(* CODESYS project MQTT 1.1.0.4.library
   Description: MQTT Stuff
      Using some cool stuff of OSCAT libs.
      see oscat.de
      
      more to describe
   Version: 1.1.0.4
   Title: MQTT
   Author: Stefan Dreyer
   DocFormat: reStructuredText
   Placeholder: SD_MQTT
   LanguageModelAttribute: qualified-access-only
   DefaultNamespace: SD_MQTT
   Company: Stefan Dreyer

Project tree, tasks and I/O mapping:
  libraries: Standard, * (System); Time and Date, 3.5.7.0 (3S - Smart Software Solutions GmbH); 3S Storage, 3.5.13.0 (3S - Smart Software Solutions GmbH); SysMem, 3.5.12.0 (System); SysTypes2 Interfaces, 3.5.4.0 (System); CmpErrors2 Interfaces, 3.5.15.0 (System); CAA Memory, 3.5.12.0 (CAA Technical Workgroup); BASIC, 3.5.16.0 (OSCAT); Common Helper for development, 1.0.0.2 (Stefan Dreyer); NETWORK, * (OSCAT)
  MQTT/
    Function Blocks/
      function block HANDLE_MQTT [ST]: ResetPingTime, MakePingPaket, StateMashineOut, StateMashineIn, BuildPublishPaket, MoveBufferForSplitPaket, BuildSubscribePaket, BuildUnsubscribePaket, SendOutData, SendInData, ParseIncoming, ParseIncomingPublish, CheckLenghtBuffer, FB_Exit, destroy, OutputPublish, MergeSplitedPublish, Publish, PublishSendDone, PushError
      function block MQTT_CONTROL [ST]
      function block MQTTPublish [ST]
      function block MQTTBase [ST]: SetMqttInOut
      function block MQTTSubscribe [ST]
      function block InsertSplitTopic [ST]: reset
      function block HandleSplitTopic [ST]: FullInit, LowInit, destroy, GetSplitTopic, FB_Exit, NewTopic, PushSplitLevel, DestroyOldSplit, CheckTopicMatchToMe, CheckTopicValid
      function block InsertSplitPayload [ST]: reset
      function block MQTTValue [ST]: Init
      function block MQTTState [ST]: Init
      function block MQTTPushover [ST]
      CallbackFBs/
        SingelCallbacks/
          function block SingelStringCallback [ST]: PublishReceived, Init, ResetReceived
          function block AllValuesCallback [ST]: PublishReceived, Init, ResetReceived
        ListCallbacks/
          function block ListStringCallback [ST]: PublishReceived, InitAsSplitTopic, InitAsSplitPayload
          function block ListAllValuesCallback [ST]: PublishReceived, InitAsSplitTopic, InitAsSplitPayload
        Callback Collector/
          function block CallbackCollector [ST]: put, PublishReceived, destroy, FB_Exit
          function block ReceiveValueWithStrucur [ST]: InitReceiveStructur
          function block ReceiveValue [ST]: PublishReceived, initAsFindPayload, initAsFindTopic, makePointer, initAsFindTopicAndPayload, SetOutput, initAsFindLastTopic
          function block ReceiveString [ST]: PublishReceived, initAsFindTopic, initAsFindPayload
          function block ReceiverBase [ST]: init, CheckMatch, GetValue
    Function/
      function InsertStringToBufferAndLength [ST]
      function DoRemainingLength [ST]
      function GetRemainingLength [ST]
      function CheckTopicLevel [ST]
      function DoRemainingLengthBevor [ST]
      function InitMQTTValue [ST]
    Structs/
      data type MQTT_IN_OUT
      data type DATA_FROM_BROKER
      data type MQTT_INFO
      data type MQTT_COM
      data type DATA_TO_BROKER
      data type MQTT_IN_DATA
      data type PAKET_DATA
      data type MQTT_OUT_DATA
      data type REMAINING_LENGTH_RETURN
      data type SPLIT_TOPIC
      data type SEND_INFOS
      data type RECEIVE_PAKET
      data type COM_CONFIG
      data type PUSHOVER_DATA
      CallbackStuff/
        data type MQTT_SUBSCRIBE_CALLBACKS
        data type LIST_STRING_CALLBACK_DATA
        data type CALLBACK_DATA
        data type LIST_ALLVALUES_CALLBACK_DATA
        data type CALLBACK_INSTANCES
      data type ONE_ERROR
    ENUMs/
      data type MESSAGETYPE
      data type QoS
      data type STEPS_OUT
      data type STEPS_IN
      data type INSERT_SPLIT_RETURN
      data type TOPIC_VALID
      data type TOPIC_MATCH
      data type PROG_NUM
      data type PUSHOVER_SOUND
      data type ERRORS
      data type RECEIVER_INIT_TYPS
      data type RECEIVE_TYPS
    Global Constants/
      global variables MyConstants
    global variables GVL_MQTT
    TestCases/
      function block TestcaseCheckTopivValid [ST]
      function block TestSubscribeOld [ST]
      function block TestMqtt [ST]
      function block TestMqttTLS [ST]
      function block TestTopicMatch [ST]
      function block TestPublishValue [ST]
      function block testHighReceive [ST]
      function block testHighReceiveSplitPayload [ST]
      function block HighLoadPublish [ST]
      function block testHighLoadPublish [ST]
      Test Interfaces/
        function block FooBarReceivingFB [ST]: PublishReceived, initAsFindTopic, getLastTreeName, initAsFindPayload
        function block exampleForFbs [ST]
        function block TestCallbackCollecktor [ST]: FB_Exit
      function block TestLongPublish [ST]
      function block TestLongStringList [ST]
      function block TestStringPointer [ST]
      function block TestUserPassword [ST]
      function block TestMemHandle [ST]
      function block TestSplitTopic [ST]
      function block testLongTime [ST]
    Docs/
      program Doku [ST]
    Exampels/
      function block TestOutOfTheBoxNoTLS [ST]
      function block TestOutOfTheBoxTLS [ST]
    Interfaces/
      interface MQTT_SUBSCRIBE_CALLBACK: PublishReceived
*)

// MQTT/Structs/MQTT_IN_OUT
TYPE MQTT_IN_OUT :
STRUCT
	//pointer to handle FB
	handleFB:POINTER TO HANDLE_MQTT;
	In: POINTER TO PAKET_DATA;
	//in free, true if free
	InFree: BOOL := TRUE;
	//time, date, impulse...
	TDI : CommonTypesAndFunctions.TIME_DATE_IMPULS_DATA;
	//TLS stuff data
	TLS_CONFIG : POINTER TO CommonTypesAndFunctions.TLS_CONFIG := 0;
	
	BROKER_CONNECTED:BOOL;
	//config for boot up
	COM_CONFIG:COM_CONFIG;
	(*client ID, only chars 0123456789abcdefghijklmnopqrstuvwxyzABCDEFGHIJKLMNOPQRSTUVWXYZ"
	System never can be anonymos
	*)
	ClientID:STRING(23):='CODESYS_MQTT';
	BuildWillTopicAndMessage: BOOL := TRUE;
	WillTopicBase:STRING(255) := 'MQTTWill';
	ClientWillTopic:STRING(255) := 'DEAD';
	ClientWillMessage:STRING(30) := 'DIED';
	//usage of dynamic RAM
	dynMemUsage:UDINT;
	{info 'TODO implement!'}
	(*set this to one if you want the client to act like the standardt says
	if set to one and we receve mor publish pakets than we can handle, QoS 0 packets are lost
	and QoS 1 and 2 packets have to be repeaded by he broker*)
	disconnectOnBufferOverflow:BOOL;
	//do you want the Reorderevents in the history?
	putReordersInHistory:BOOL := FALSE;
	//Log buffer Moves?
	LogBufferMoves:BOOL;
END_STRUCT
END_TYPE

// MQTT/ENUMs/MESSAGETYPE
TYPE MESSAGETYPE :
(
	CONNECT 	:= 16#10,
	CONNACK 	:= 16#20,
	PUBLISH 	:= 16#30,
	PUBACK 		:= 16#40,
	PUBREC		:= 16#50,
	PUBREL		:= 16#60,
	PUBCOMP		:= 16#70,
	SUBSCRIBE 	:= 16#80,
	SUBACK 		:= 16#90,
	UNSUBSCRIBE := 16#A0,
	UNSUBACK 	:= 16#B0,
	PINGREQ 	:= 16#C0,
	PINGRESP	:= 16#D0,
	DISCONNECT 	:= 16#E0
) BYTE;
END_TYPE

// MQTT/ENUMs/QoS
TYPE QoS :
(
	AtMostOnce:= 2#0,
	AtLeastOnce:= 2#1,
	ExactlyOnce:= 2#10,
	Fail:=2#10000000
) BYTE;
END_TYPE

// MQTT/Structs/DATA_FROM_BROKER
TYPE DATA_FROM_BROKER :
STRUCT
	//use array in size of network buffer to split message dynamic, maybe not ... best is dynamic mammory....
	//or use an array of Pointer....
	//or callbacks
	// so lets try to buffer public messages and releas one per cycle to application...
	//now we try dynamic memmory....
	//MQTT Topic from Broker
	MqttTopic:POINTER TO STRING;
	Topics:POINTER TO SPLIT_TOPIC;
	//MQTT Payload for Broker
	//Payload from broker --> Pointer
	MqttPayload:POINTER TO BYTE;
	//Payload size
	MqttPayloadSize:UDINT;
	//MQTT Message Type
	MessageType:MESSAGETYPE;
	//Data received
	DataReceived:BOOL;
	
END_STRUCT
END_TYPE

// MQTT/Structs/MQTT_INFO
TYPE MQTT_INFO :
STRUCT
	MQTT_CONNECTED : BOOL;
	MQTT_ERROR : STRING(OSCAT_BASIC.STRING_LENGTH);
END_STRUCT
END_TYPE

// MQTT/Structs/MQTT_COM
(*contro struct between HANDLE_MQTT and MQTT_CONTROL*)
TYPE MQTT_COM :
STRUCT
	S_BUF : NETWORK_BUFFER;
	R_BUF : NETWORK_BUFFER;
	MQTT_CON : BOOL;//if falling edge close with disconnect packet
	MQTT_ABORT :BOOL;//if using this to disconnect, don't send disconnect paket....
	MQTT_URL : STRING(OSCAT_BASIC.STRING_LENGTH);
	MQTT_PACKET_NO : WORD;
	TIMEOUT : TIME;
	//DNS_IP4 : DWORD;
	//set to true if you want to use TLS
	TLS: BOOL;
	//data to TLS stuff
	TLS_CONFIG:POINTER TO CommonTypesAndFunctions.TLS_CONFIG := 0;
	(*
	0= non
	1= received
	2= error*)
	MQTT_RCV_STATE : BYTE;
	ERROR_C : DWORD;
	ERROR_T : BYTE;
	//CONNECT_TO_LOCALHOST:BOOL;
	CLIENT_ID:STRING(23);
	CLIENT_WILL_TOPIC:STRING(255);//Topic vof will message after client id
	CLIENT_WILL_MESSAGE_DEAD:STRING(255);
	{info 'implement parameter'}
	CLIENT_WILL_RETAIN:BOOL:=TRUE;
	//pakte wihout request-- return to receive state 1
	MQTT_NO_AWNSER: BOOL;


END_STRUCT
END_TYPE

// MQTT/Structs/DATA_TO_BROKER
TYPE DATA_TO_BROKER :

STRUCT
	//Data of Paket
	PaketData:PAKET_DATA;
END_STRUCT
END_TYPE

// MQTT/Structs/MQTT_IN_DATA
TYPE MQTT_IN_DATA :
STRUCT
	step:STEPS_IN;
	PaketID:WORD;
	WaitsForBuffFree:ULINT;
	TimeOut:ton;
	TimeOutStarted:BOOL;
	PUBLISHOrder:UINT;
	PUBCOMPOrder:UINT;
	QoS:QoS;
	CountPubrecRepeat:UINT;;
END_STRUCT
END_TYPE

// MQTT/Structs/PAKET_DATA
TYPE PAKET_DATA :
STRUCT
	//MQTT Topic for Broker
	MqttTopic:POINTER TO STRING;
	//Topic length
	MqttTopicLength:UINT;
	//MQTT Payload for Broker
	MqttPayload:POINTER TO BYTE;
	//Payload length
	MqttPayloadLength:UDINT;
	//MQTT Message Type
	MessageType:MESSAGETYPE;
	//MQTT QoS
	MessageQoS:QoS;
	//SUCACK QoS Response
	SubackQoS:QoS;
	//MQTT reatin
	MessageRetain:BOOL;
	//Retry of paket
	DUP: BOOL;
	//PakatID for header
	PaketId:WORD;
	//ID of MQTT FB to store or of request to Broker
	//FbId:UINT;
	//Send was succsessfull
	SendSucsess: BOOL;
	//Callback FB for subscription
	Callback:MQTT_SUBSCRIBE_CALLBACK;
	//split topic for subscribe
	SplitTopic:POINTER to HandleSplitTopic; 
	//errore registering the callback
	CallbackError: BOOL;
	//Expecting String
	ExpectingString: BOOL;


	
END_STRUCT
END_TYPE

// MQTT/Structs/MQTT_OUT_DATA
TYPE MQTT_OUT_DATA :
STRUCT
	InDataFromFb: POINTER TO PAKET_DATA;
	step:STEPS_OUT;
	WaitsForBuffFree:ULINT;
	PUBRECOrder:UINT;
	TimeOut:ton;
	TimeOutStarted:BOOL;
	PUBLISHOrder:UINT;
	PUBRELRepeatCounter:UINT;
END_STRUCT
END_TYPE

// MQTT/ENUMs/STEPS_OUT
{attribute 'qualified_only'}
{attribute 'strict'}
TYPE STEPS_OUT :
(
	WAIT_DATA := 0, SEND_PUBLSIH, WAIT_PUBREC, SEND_PUBREL,
	WAIT_PUBCOMP, WAIT_PUBACK, WAIT_PINGRESP, SEND_SUBSCRIBE, 
	WAIT_SUBACK, SEND_UNSUBSCRIBE, WAIT_UNSUBACK
);
END_TYPE

// MQTT/ENUMs/STEPS_IN
{attribute 'qualified_only'}
{attribute 'strict'}
TYPE STEPS_IN :
(
	WAIT_DATA := 0, SEND_PUBACK, SEND_PUBREC, 
	WAIT_PUBREL, SEND_PUBCOMP
);
END_TYPE

// MQTT/Structs/REMAINING_LENGTH_RETURN
TYPE REMAINING_LENGTH_RETURN :
STRUCT
	RemainingLength:UDINT;
	IndexAfterRemainingLength:UINT; 
	Error:BOOL;
	//not all bytes of remaining length in buffer...
	BuffToSmall:BOOL;
	//size of remaining length
	SizeRemainingLength:USINT;
	
END_STRUCT
END_TYPE

// MQTT/Structs/SPLIT_TOPIC
TYPE SPLIT_TOPIC :
STRUCT
	//this is going to be a pointer to a array of pointer to stings  
	Topics:POINTER TO POINTER TO STRING;
	//count of vailid fields in the array
	ValidFields:UINT;
	
END_STRUCT
END_TYPE

// MQTT/ENUMs/INSERT_SPLIT_RETURN
{attribute 'qualified_only'}
{attribute 'strict'}
TYPE INSERT_SPLIT_RETURN :
(
	INSERT_NOT_VALID := 0, INSERT_DONE , INSERT_PENDING, INSERT_ERROR
);
END_TYPE

// MQTT/ENUMs/TOPIC_VALID
{attribute 'qualified_only'}
{attribute 'strict'}
TYPE TOPIC_VALID :
(
	TOPIC_UNTESTED := 0, TOPIC_VALID := 2, TOPIC_NOT_VALID := 1, TOPIC_NO_TEST := 3
)BYTE;
END_TYPE

// MQTT/ENUMs/TOPIC_MATCH
{attribute 'qualified_only'}
{attribute 'strict'}
TYPE TOPIC_MATCH :
(
	TOPIC_MATCHES := 1, TOPIC_DONT_MATCHES := 2, TOPIC_NO_MEMORY := 3
)BYTE;
END_TYPE

// MQTT/Structs/SEND_INFOS
TYPE SEND_INFOS :
STRUCT
		
//this index is to be subscribed
	SubscribeIndex:UINT;
	SubscribeNeeded:BOOL := FALSE;
	SubscribeBlocking: BOOL;

	//this index is to be subscribed
	
	UnsubscribeIndex:UINT;
	UnsubscribeNeeded:BOOL := FALSE;
	UnsubscribeBlocking: BOOL;

	//this index is to be published
	PublishBlocking: BOOL;
	PublishBlockingIndex : UINT;

	//this index is to be published
	PingIndex:UINT;
	PingNeeded: BOOL;
	
END_STRUCT
END_TYPE

// MQTT/Structs/RECEIVE_PAKET
//used for test cases...
TYPE RECEIVE_PAKET :
STRUCT
	//MQTT Topic
	MqttTopic:STRING(2000);
	//MQTT Payload
	MqttPayload:STRING(2000);
END_STRUCT
END_TYPE

// MQTT/ENUMs/PROG_NUM
{attribute 'qualified_only'}
{attribute 'strict'}
TYPE PROG_NUM :
(
	Publish, Subscribe, ParseIncomming, MoveBuffer, ParsePublish, GetBufferFreePos, GetSplitTopic, DESTROY_HANDLE_MQTT,
	DESTROY_SPLIT_TOPIC, STATE_MASHINE_IN,  STATE_MASHINE_OUT, SendOutData, SendInData, SendOutDataInsertTopic, SendOutDataInsertPayload,
	DESTROY_SPLIT_TOPIC_DONE, DESTROY_HANDLE_MQTT_DONE, DESTROY_CALLBACK_COLLECTOR, DESTROY_CALLBACK_COLLECTOR_DONE
);
END_TYPE

// MQTT/Structs/COM_CONFIG
(*here the maximum sizes of paylod and topics are defined
if dynamic low init of split topic is used, don't care about MaxTopicElementSize*)
TYPE COM_CONFIG :
STRUCT
	//max payload size
	MaxPayloadSize : UDINT := 2000;
	//max topic levels
	MaxTopicLevels:UINT := 25;
	//Max Topic elemt size
	MaxTopicElementSize:UINT:=255;
	
END_STRUCT
END_TYPE

// MQTT/Structs/PUSHOVER_DATA
TYPE PUSHOVER_DATA :
STRUCT
	Trigger:POINTER TO BOOL;
	Topic:POINTER TO STRING;
	Payload:POINTER TO STRING;
	Prio:USINT;
	Sound:PUSHOVER_SOUND;
	IsConfig:BOOL;
	R_T:R_TRIG;
	NeedToPush:BOOL;
	Negate:BOOL;
END_STRUCT
END_TYPE

// MQTT/ENUMs/PUSHOVER_SOUND
{attribute 'qualified_only'}
{attribute 'strict'}
TYPE PUSHOVER_SOUND :
(
	Standart := 1
);
END_TYPE

// MQTT/Structs/CallbackStuff/MQTT_SUBSCRIBE_CALLBACKS
TYPE MQTT_SUBSCRIBE_CALLBACKS :
STRUCT
	Callback:MQTT_SUBSCRIBE_CALLBACK;
	//expecting string
	ExpectingString: BOOL;
	SplitTopic:POINTER TO HandleSplitTopic;
	//set to false if slot is aquired by an subscription
	free:BOOL:=TRUE;
	
END_STRUCT
END_TYPE

// MQTT/Structs/CallbackStuff/LIST_STRING_CALLBACK_DATA
TYPE LIST_STRING_CALLBACK_DATA :
STRUCT
	//pointer to target string
	Target:POINTER TO STRING;
	//pointer to last subtopic or Payload Data to compare with
	SubTopic:POINTER TO STRING;

END_STRUCT
END_TYPE

// MQTT/Structs/CallbackStuff/CALLBACK_DATA
(*this data is passed to a subscription callback*)

TYPE CALLBACK_DATA :
STRUCT
	{info 'make size check due use of memmove...'}
	(*the Payload String,
	be aware, this pointer will only copy 255 bytes. If more needed, use memmove!*)
	PayloadString:POINTER TO STRING(255);
	(*pointer to binary payload*)
	Payload:POINTER TO BYTE;
	(*size of binary payload*)
	PayloadSize:UDINT;
	(*here you get the compleete received topic string, maybe bigger then 255 byte!*)
	TopicOut:POINTER TO STRING(255);
	//split topic....
	TopicOutSplit:POINTER TO SPLIT_TOPIC;
	//Payload is string
	PayloadIsString: BOOL;

END_STRUCT
END_TYPE

// MQTT/Structs/CallbackStuff/LIST_ALLVALUES_CALLBACK_DATA
TYPE LIST_ALLVALUES_CALLBACK_DATA :
STRUCT
	VarTYPE:CommonTypesAndFunctions.VAR_TYPES;
	Target:CommonTypesAndFunctions.ALL_TYPES_UNION_POINTER;
	//pointer to last subtopic or Payload Data to compare with
	SubTopic:POINTER TO STRING;
END_STRUCT
END_TYPE

// MQTT/Structs/CallbackStuff/CALLBACK_INSTANCES
{attribute 'enable_dynamic_creation'} 
TYPE CALLBACK_INSTANCES :
STRUCT
	callback:MQTT_SUBSCRIBE_CALLBACK;
	next: POINTER TO CALLBACK_INSTANCES := 0;
	

END_STRUCT
END_TYPE

// MQTT/Structs/ONE_ERROR
TYPE ONE_ERROR :
STRUCT
	error:ERRORS;
	when:DT;
	ERROR_C : DWORD;
	ERROR_T : BYTE;
	text:STRING(255);
	MqttsDoneIo:ULINT;
	SendetBytes:ULINT;
	ReceivedBytes:ULINT;
END_STRUCT
END_TYPE

// MQTT/ENUMs/ERRORS
{attribute 'qualified_only'}
{attribute 'strict'}
TYPE ERRORS :
(
	NOT_VALID := 0,
	CONNECTION_REFUSED := 1, MAX_PING_REPEATS := 2,
	RECEIVED_PUBISH_TO_BIG_FOR_BUFFER := 3, FULL_PACKET_NOT_RECEIVED := 4,
	RECEIVED_PUBLISH_REMAINING_LENGTH_ERROR := 5,
	NO_MORE_RECEIVE_SLOTS_FREE := 6,
	CONNECTION_ESTABLISHED := 7, TIMEOUT_CONNECTION := 8,
	REPEAT_PUBLISH_PUBCOMP := 9, REPEAT_PUBREL := 10, 
	REORDER_PUBREC := 11, REORDER_PUBLISH_OUTGOING := 12,
	REPEAT_PUBLISH_PUBREC := 13, REPEAT_PUBLISH_PUBACK := 14,
	HARD_DISCONNECT := 15, MOVED_TO_BIG_RECEIVE_BUFFER := 16,
	NEED_BUFFER_MOV := 17, UNKNOWN_PAKET_RECEIVED := 18,
	TO_BIG_PAKET := 19, TOPIC_MOVED_DOWN := 20,
	TOPIC_AND_PAYLOAD_MOVED := 21, PAYLOAD_MOVED_UP := 22,
	TOPIC_MOVED_DOWN_NETWORK := 23, PAYLOAD_MOVED_UP_NETWORK := 24,
	REPEAT_PUBREC := 25, PUBREC_DISCHARGE := 26,
	REODER_PUBLISH_INCOMMING := 27, REORDER_PUBCOMP := 28,
	UNKNOWN_PAKET_IN_MQTT_IN_OUT := 29,
	PUBLISH_NO_SLOT_FREE := 30, OUT_OFF_DYN_MEMORY := 31
);
END_TYPE

// MQTT/ENUMs/RECEIVER_INIT_TYPS
{attribute 'qualified_only'}
{attribute 'strict'}
TYPE RECEIVER_INIT_TYPS :
(
	(*searching for full matching topic*)
	FIND_FULL_TOPIC := 0,
	(*searching for match of last topic*) 
	FIND_LAST_TOPIC,
	(*searching on paylod, from start, spared with delimiter*) 
	FIND_PAYLOAD,
	(*search full topic and one JSON element*)
	JSON_FULL,
	(*searching for last topic and one JSON element*)
	JSON_SMALL,
	(*search with MQTT string(including +, #)*)
	MQTT_STRING,
	(*search with MQTT string(including +, #), then JSON*)
	MQTT_STRING_JSON
);
END_TYPE

// MQTT/ENUMs/RECEIVE_TYPS
{attribute 'qualified_only'}
{attribute 'strict'}
TYPE RECEIVE_TYPS :
(
	FIND_PAYLOAD := 0, FIND_TOPIC := 1, FIND_LAST_TOPIC := 2, FIND_LAST_TOPIC_AND_PAYLOAD := 3 
);
END_TYPE

// MQTT/Global Constants/MyConstants
{attribute 'qualified_only'}
VAR_GLOBAL CONSTANT
	//count of simultanus packets workt on
	IN_OUT_SLOTS_SIZE:UINT:=50;
	NETWORK_BUFFER_LONG_SIZE:UINT:=4095;
	KEEP_ALIVE_TIME : DWORD := 8;
	SENDING_TIMEOUT : TIME := T#4S;
	REPEAT_TIMEOUT : TIME := T#2S;
	REORDER_VALUE :UINT:=50000;//50000
	SUBSTRACTION_VALUE:UINT:=30000;//20000
	MAX_PUBREL_REPEATS : UINT :=10;
END_VAR

// MQTT/GVL_MQTT
{attribute 'qualified_only'}
VAR_GLOBAL
	//Last Progamm stat for debug timeout exception
	ProgNum:PROG_NUM;
	//LOG_BUFFER_MOVES:BOOL;
END_VAR

// MQTT/Function Blocks/HANDLE_MQTT
(*
var/log/mosquitto/mosquitto.log
Messsages are not beeing repeatet, if timout for an answer then connection is canceled, new established and the publisher have to start new
Start the command line subscriber:
mosquitto_sub -v -t 'test/topic'
mosquitto_sub -v -h test.mosquitto.org -t 'test/topic'


sudo apt-get install tshark 

tshark -i 1 -a duration:60 -w /tmp/wlan.pcap

debug / logging :
mosquitto_sub -v -t '$SYS/#'
sudo nano /etc/mosquitto/mosquitto.conf  --> 'log_type all'
Publish test message with the command line publisher:
mosquitto_pub -t 'test/topic' -m 'helloWorld'
change check free to InFbNo

kopieren
sudo cp /var/log/mosquitto/mosquitto.log /tmp/
zugriff
sudo chmod -v a=r /tmp/mosquitto.log


TODO: Take care of clean session, is enabled, do it paramable?
	
*)


FUNCTION_BLOCK HANDLE_MQTT  
VAR_IN_OUT
	
	MQTT_IN_OUT:MQTT_IN_OUT;
END_VAR
VAR_INPUT
	ENABLE : BOOL;
	//use format: user:password@domain:port
	URL : STRING(OSCAT_BASIC.STRING_LENGTH);
	TIMEOUT : TIME;
	TLS: BOOL;

END_VAR
VAR_OUTPUT
	ERROR_C : DWORD;
	ERROR_T : BYTE;
END_VAR
VAR
	MQTT_INFO : MQTT_INFO;
	DT_MQTT:CommonTypesAndFunctions.TIME_DATE_IMPULS;
	MQTT_CONTROL: MQTT_CONTROL;
	step : INT;
	i1 : UINT;
	
	PingSlot:UINT;
	
	COM: MQTT_COM;
	
	connected: BOOL;

	TimeoutConnection:TON;
		
	MqttsDoneIo:ULINT;
	
	CycleTime:DWORD;
	LastCycleTime:DWORD;
	NextPingTime:CAA.TICK;
	PingTime : CAA.TICK := (MyConstants.KEEP_ALIVE_TIME * 1000) - 6000;//next ping after 6 seconds 
	// Ping was sendet
	PingRequestet: BOOL;
	PingData:DATA_TO_BROKER;
	myFbNo:UINT;
	PubrelOrderIndexCounter:UINT;
	PubcompOrderIndexCounter:UINT;
	
	
	
	//Slots for state masdchien for outgoing packets(to broker)
	OutDataSlots:ARRAY[0..MyConstants.IN_OUT_SLOTS_SIZE] OF MQTT_OUT_DATA;
	//Slots for state masdchien for incomming packets(from broker)
	InDataSlots:ARRAY[0..MyConstants.IN_OUT_SLOTS_SIZE] OF MQTT_IN_DATA;
	PublishSendListCount:UINT;
	PublishSendList:ARRAY[0..MyConstants.IN_OUT_SLOTS_SIZE] OF UINT;
	PubrelSendListCount:UINT;
	PubrelSendList:ARRAY[0..MyConstants.IN_OUT_SLOTS_SIZE] OF UINT;
	PubackSendListCount:UINT;
	PubackSendList:ARRAY[0..MyConstants.IN_OUT_SLOTS_SIZE] OF UINT;
	PubrecSendListCount:UINT;
	PubrecSendList:ARRAY[0..MyConstants.IN_OUT_SLOTS_SIZE] OF UINT;
	PubcompSendListCount:UINT;
	PubcompSendList:ARRAY[0..MyConstants.IN_OUT_SLOTS_SIZE] OF UINT;
	
	//Repeted Publishs
	RepeatedPublish:ULINT;
	//Repeatet publishs afert ot much repeat of pubrel
	RepeatedPublishsAfterPubrel:ULINT;
	//Repeted pubrel
	RepeatedPubrel:ULINT;
	//Repeted Ping
	CountRepeatedPing:ULINT;
	//Repeated pings untill disconnect
	CountRepeatedPingDisconnect:UINT;
	//count of Publishs unacknowledged
	PublishsUnacknowledged:UINT;
	//last part of 255 chars of to big paket topic
	LastToBigTopic:STRING(255);
	//count of to big topics
	CountToBigTopics:ULINT;
	//Cont of ength Error Pakets
	CountLengthErrors:ULINT;
	//Count of repeatet publishs
	CountRepeatPublishReceive:ULINT;
	//Count Received Publishs
	CountReceivedPublishs:ULINT;
	//count sended publishs
	CountSendedPublishs:ULINT;
	//Count of repeated subscribs
	CountRepeatSubscribe:ULINT;
	//Count of repeated unsubscribs
	CountRepeatUnsubscribe:ULINT;
	//Count of repeatet pubrec
	CountRepeatetPubrec:ULINT;
	//Count of OutputPublish calls
	CountOutputPublishCalled:ULINT;
	PUBREC_ERROR_ID_BUFFER:ARRAY[0..PUBREC_ERROR_ID_BUFFER_SIZE -1] OF UINT;
	PUBREC_ERROR_INDEX:UINT;
	//send Publish order Index
	OutgoingPublishOrderIndexCounter:UINT;
	//receive Publish order Index
	IncomingPublishOrderIndexCounter:UINT;
	//Received Pubrel, Paket not found
	CountReceivePubrelUnknown:ULINT;
	//Received Unsuback, Paket not found
	CountReceiveUnsubackUnknown:ULINT;
	//Received Suback, Paket not found
	CountReceiveSubackUnknown:ULINT;
	//Received Puback, Paket not found
	CountReceivePubackUnknown:ULINT;
	//Received Pubrec, Paket not found
	CountReceivePubrecUnknown:ULINT;
	//Received Pubcomp, Paket not found
	CountReceivePubcompUnknown:ULINT;
	SendInfos:SEND_INFOS;
	CountOutSendNotFree:ULINT;
	CountInSendNotFree:ULINT;
	CountCantSendPublishBufferToFull:ULINT;
	CounterPublishSendForMonitor:UINT;
	PublishsSendPerSeconde:UINT;
	CounterPublishReceivedForMonitor:UINT;
	PublishsReceivedPerSeconde:UINT;
	NotKnownPaket:MESSAGETYPE;
	CountUnkownPaket:ULINT;
	LastPaktetForUnkownPaket:MESSAGETYPE;
	HelperLastPaktetForUnkownPaket:MESSAGETYPE;
	CountBufferMoves:ULINT;
	CountNothingSend:ULINT;
	CountConnectAttempt:ULINT;
	//count of topic size exceeded
	CountSplitTopicSizeExceeded:ULINT;
	
	
	CountWaitForRestOfPaket:ULINT;
	CountResetBufferIn:ULINT;
	InBufferMoved:UINT;
	SendFree: BOOL;
	
	MySplitTopic:HandleSplitTopic;
	
	
	InsertSplitTopic:InsertSplitTopic;
	InsertSplitPayload:InsertSplitPayload;
	StepBuildPublish:INT;
	StepBuildSubscribe:INT;
	StepBuildUnsubscribe:INT;
	//use this buffer for received publish packets whos size exceded network buffer Size
	SplitPublishBuffer:POINTER TO BYTE;
	SplitPublishBufferSize:UDINT;
	SplitPublishLength:UDINT;
	//output from buffer Don't write new data!
	MaxPublishPacketSize:UDINT;
	PayloadMemorySize: DWORD;
	
	SubscribeCallbacks:ARRAY[0..CALLBACKS_BUFFER_SIZE - 1] OF MQTT_SUBSCRIBE_CALLBACKS;
	
	TopicMemorySize: DWORD;
	
	COM_CONFIG:COM_CONFIG;

	//publish paket broken, waiting for more data
	PublishSplited: BOOL;
	DoDisconnect: BOOL;
	SendetBytes:ULINT;
	ReceivedBytes:ULINT;
	InSlotsWorking:UINT;
	OutSlotsWorking:UINT;
	SplitPublishBufferAllocationSize:UDINT;
	DynMemUsagePointer : POINTER TO UDINT;
	//callbacks array full
	CallbacksFull: BOOL;

	ErrorHistory:ARRAY[0..COUNT_ERROR_HISTORY]OF ONE_ERROR;
	
	localTdi:CommonTypesAndFunctions.TIME_DATE_IMPULS_DATA;
	
	//Step 10 Init is done:
	StepInitDone: BOOL;

	//Local copy of log buffer moves
	LogBufferMoves: BOOL;

	
END_VAR

VAR CONSTANT
	{info 'make configurable'}
	CALLBACKS_BUFFER_SIZE:UINT:=200;
	RECEIVE_PUBLISH_BUFFER_SIZE : UINT := NETWORK_BUFFER_LONG_SIZE * 2;
	TRANSMIT_BUFFER_SIZE : UINT := NETWORK_BUFFER_LONG_SIZE;
	SIZE_PUBREL:UINT := 4;
	SIZE_UNSUBACK:UINT := 4;
	SIZE_PINGRESP:UINT := 2;
	SIZE_PINGREQ:UINT := 2;
	SIZE_SUBACK:UINT := 5;
	SIZE_PUBACK:UINT := 4;
	SIZE_PUBREC:UINT := 4;
	SIZE_PUBCOMP:UINT := 4;
	SIZE_PAKET_BUFFER_HEADER:UINT := 4;
	PUBREC_ERROR_ID_BUFFER_SIZE:UINT:=100;
	MAX_PING_REPEATS:UINT:=10;
	SPLIT_PUBLISH_BUFFER_ADDITIONAL_RAM:UINT:=17;
	COUNT_MAX_PUBREC_REPEAT_TO_DISCHARGE:UINT:=20;
	COUNT_ERROR_HISTORY:UINT:=1000;
END_VAR

IF MQTT_INFO.MQTT_CONNECTED THEN
	SendFree := COM.S_BUF.SIZE = 0;	
END_IF

LogBufferMoves := MQTT_IN_OUT.LogBufferMoves;

CycleTime := OSCAT_BASIC.T_PLC_MS() - LastCycleTime;
LastCycleTime := OSCAT_BASIC.T_PLC_MS();
//get system time and so one
DT_MQTT(
	TDI_Data:= MQTT_IN_OUT.TDI);
localTdi:= MQTT_IN_OUT.TDI ; 
TimeoutConnection(IN:= step = 10, PT:= T#5S);

CASE step OF

	00:	MQTT_IN_OUT.BROKER_CONNECTED := FALSE;
		IF ENABLE THEN
			MQTT_IN_OUT.handleFB := THIS;
			PingRequestet := FALSE;
			PublishsUnacknowledged := 0;
			PUBREC_ERROR_INDEX := 0;
			CountRepeatedPingDisconnect := 0;
			SendetBytes := 0;
			ReceivedBytes := 0;		
			PublishSplited := FALSE;
			DoDisconnect := FALSE;
			SendInfos.PingNeeded := FALSE;
			SendInfos.SubscribeNeeded := FALSE;
			SendInfos.UnsubscribeNeeded := FALSE;
			StepBuildPublish := 0;
			StepBuildSubscribe := 0;
			StepBuildUnsubscribe := 0;
			InsertSplitTopic.reset();
			InsertSplitPayload.reset();
			CountConnectAttempt := CountConnectAttempt + 1;
			DynMemUsagePointer := ADR(MQTT_IN_OUT.dynMemUsage);
			COM.MQTT_URL := URL;
			COM.TIMEOUT := TIMEOUT;
			COM.CLIENT_ID := MQTT_IN_OUT.ClientID;
			COM.TLS := TLS;
			COM.TLS_CONFIG := MQTT_IN_OUT.TLS_CONFIG;
			ResetPingTime();
			//build will topic
			IF MQTT_IN_OUT.BuildWillTopicAndMessage THEN
				COM.CLIENT_WILL_TOPIC := MQTT_IN_OUT.WillTopicBase;
				COM.CLIENT_WILL_TOPIC := Standard.CONCAT(STR1:= COM.CLIENT_WILL_TOPIC, '/');
				COM.CLIENT_WILL_TOPIC := Standard.CONCAT(STR1:= COM.CLIENT_WILL_TOPIC, STR2:= COM.CLIENT_ID);
				COM.CLIENT_WILL_TOPIC := Standard.CONCAT(STR1:= COM.CLIENT_WILL_TOPIC, '/');
				COM.CLIENT_WILL_TOPIC := Standard.CONCAT(STR1:= COM.CLIENT_WILL_TOPIC, MQTT_IN_OUT.ClientWillTopic);
				COM.CLIENT_WILL_TOPIC := Standard.CONCAT(STR1:= '/', COM.CLIENT_WILL_TOPIC);
				COM.CLIENT_WILL_TOPIC := Standard.CONCAT(STR1:= COM.CLIENT_ID, COM.CLIENT_WILL_TOPIC);
			ELSE
				COM.CLIENT_WILL_TOPIC := MQTT_IN_OUT.ClientWillTopic;
			END_IF
			COM.CLIENT_WILL_MESSAGE_DEAD := MQTT_IN_OUT.ClientWillMessage;
			COM_CONFIG := MQTT_IN_OUT.COM_CONFIG;
			FOR i1 := 0 TO MyConstants.IN_OUT_SLOTS_SIZE - 1 DO
				//reset in slots
				InDataSlots[i1].step := STEPS_IN.WAIT_DATA;
				OutDataSlots[i1].step := STEPS_OUT.WAIT_DATA;
				//reset Timeouts...
				InDataSlots[i1].TimeOutStarted := FALSE;
				OutDataSlots[i1].TimeOutStarted := FALSE;
				InDataSlots[i1].TimeOut(IN:= InDataSlots[i1].TimeOutStarted, PT:= MyConstants.REPEAT_TIMEOUT);
				OutDataSlots[i1].TimeOut(IN:= OutDataSlots[i1].TimeOutStarted, PT:= MyConstants.REPEAT_TIMEOUT);
			END_FOR
			//reset callbacks
			FOR i1 := 0 TO CALLBACKS_BUFFER_SIZE - 1 DO
				SubscribeCallbacks[i1].free := TRUE; 
			END_FOR
			IF  MySplitTopic.FullInit(TopicsLevelInit:= COM_CONFIG.MaxTopicLevels, SplitElementSizeInit:= COM_CONFIG.MaxTopicElementSize, dynMemUsageInit:= ADR(MQTT_IN_OUT.dynMemUsage)) THEN
				
				PayloadMemorySize := COM_CONFIG.MaxPayloadSize;
				{warning disable C0033}
				TopicMemorySize := COM_CONFIG.MaxTopicElementSize * COM_CONFIG.MaxTopicLevels;
				MaxPublishPacketSize := (COM_CONFIG.MaxTopicElementSize * COM_CONFIG.MaxTopicLevels) + PayloadMemorySize;
				SplitPublishBufferAllocationSize := MaxPublishPacketSize + SPLIT_PUBLISH_BUFFER_ADDITIONAL_RAM;
				{info 'semaphore'}
				SplitPublishBuffer  := __NEW(BYTE, SplitPublishBufferAllocationSize);//some additional bytes for paket overhead and termination
				IF SplitPublishBuffer = 0 THEN
					PushError(newError:= ERRORS.OUT_OFF_DYN_MEMORY, text:='No Dyn Memory in Step 00 in Handle' );
					step := 60;
				ELSE
					MQTT_IN_OUT.dynMemUsage := MQTT_IN_OUT.dynMemUsage + SplitPublishBufferAllocationSize;
					{warning restore C0033}
		
					step := 10;
					COM.MQTT_CON := TRUE;
					StepInitDone := TRUE;
					
				END_IF
			ELSE
				PushError(newError:= ERRORS.OUT_OFF_DYN_MEMORY, text:='No Dyn Memory in Step 00 in Handle on create SplitTopic' );
				step := 60;
			END_IF
		END_IF	
	10:	IF MQTT_INFO.MQTT_CONNECTED THEN
			step := 40;
			MQTT_IN_OUT.BROKER_CONNECTED := TRUE;
			PushError(newError:= ERRORS.CONNECTION_ESTABLISHED, text:='');
		END_IF
		IF TimeoutConnection.Q THEN
			PushError(newError:= ERRORS.TIMEOUT_CONNECTION, text:='' );
			step := 0;//reset steps
			destroy();
			
		END_IF
	40:	
		IF PublishSplited THEN
			MergeSplitedPublish(MQTT_IN_OUT:= ADR(MQTT_IN_OUT));
		END_IF	
		ParseIncoming(MQTT_IN_OUT:= ADR(MQTT_IN_OUT));
		PublishSendListCount := 0;
		PubrelSendListCount := 0;
		PubackSendListCount := 0;
		PubrecSendListCount := 0;
		PubcompSendListCount := 0;
		StateMashineIn(MQTT_IN_OUT:= ADR(MQTT_IN_OUT));
		StateMashineOut( MQTT_IN_OUT:= ADR(MQTT_IN_OUT));
		
		SendOutData(MQTT_IN_OUT:= ADR(MQTT_IN_OUT));
		SendInData(MQTT_IN_OUT:= ADR(MQTT_IN_OUT));
	
		IF MQTT_IN_OUT.TDI.IMP THEN
			PublishsSendPerSeconde := CounterPublishSendForMonitor;
			CounterPublishSendForMonitor := 0;
			PublishsReceivedPerSeconde := CounterPublishReceivedForMonitor;
			CounterPublishReceivedForMonitor := 0;
		END_IF
		IF COM.S_BUF.SIZE = 0 THEN
			CountNothingSend := CountNothingSend + 1;
		END_IF
		IF NOT ENABLE THEN 	(* beenden? *)
			step := 50;
			
		END_IF;
		IF DoDisconnect THEN
			DoDisconnect := FALSE;
			//here hard disconnect
			PushError(newError:= ERRORS.HARD_DISCONNECT , text:='');
			COM.MQTT_CON := FALSE; (* MQTT Verbindung beenden *)
			COM.MQTT_ABORT := TRUE;
			MQTT_IN_OUT.BROKER_CONNECTED := FALSE;
			step := 60;
		END_IF

(* ~~~~~~~~~~~~~~~~~~~~~~ *)

50: 
	COM.MQTT_CON := FALSE; (* MQTT Verbindung beenden *)
	MQTT_IN_OUT.BROKER_CONNECTED := FALSE;
	step := 60;//wait for disconnect
60:
	IF MQTT_INFO.MQTT_CONNECTED = FALSE THEN
		destroy();
		step := 0;
		MQTT_IN_OUT.BROKER_CONNECTED := FALSE;
	END_IF
END_CASE;



(* ########################## *)

IF CountRepeatedPingDisconnect > MAX_PING_REPEATS THEN
	DoDisconnect := TRUE;
	IF step = 40 THEN
		PushError(newError:= ERRORS.MAX_PING_REPEATS, text:='');
	END_IF
END_IF


SendetBytes := SendetBytes + COM.S_BUF.SIZE;
MQTT_CONTROL(COM:= COM, INFO:=MQTT_INFO);
ReceivedBytes := ReceivedBytes + COM.R_BUF.SIZE;
ERROR_C := COM.ERROR_C;
ERROR_T := COM.ERROR_T;
//handl ping telegram
IF NextPingTime < TICKS.GetTick(xDummy:= TRUE) AND NOT PingRequestet AND connected THEN
	
	MakePingPaket(MQTT_IN_OUT := MQTT_IN_OUT);
	
END_IF

IF COM.ERROR_T > BYTE#0 THEN  (* FEHLER *)
	DoDisconnect := TRUE;
	MQTT_IN_OUT.BROKER_CONNECTED := FALSE;
	PushError(newError:= ERRORS.CONNECTION_REFUSED, text:='');
END_IF;
//put status to local clients
 

connected := MQTT_IN_OUT.BROKER_CONNECTED;
(* ########################## *)

(* revision history


*)

METHOD ResetPingTime
VAR_INPUT
END_VAR
NextPingTime := PingTime + TICKS.GetTick(xDummy:= TRUE);
CountRepeatedPingDisconnect := 0;
END_METHOD

METHOD MakePingPaket
VAR_INPUT
END_VAR
VAR_IN_OUT
	MQTT_IN_OUT:MQTT_IN_OUT;
END_VAR
IF MQTT_IN_OUT.InFree THEN 
	MQTT_IN_OUT.IN := ADR(PingData); //set request
	PingData.PaketData.MessageType := MESSAGETYPE.PINGREQ;
	MQTT_IN_OUT.InFree := FALSE;
	PingRequestet := TRUE;
END_IF
END_METHOD

METHOD StateMashineOut
VAR_INPUT
	
	//StepData:POINTER TO MQTT_OUT_DATA;
	MQTT_IN_OUT : POINTER TO MQTT_IN_OUT;
END_VAR
VAR
	i:UINT;
	j:UINT;
	tmpLowest:UINT;
	minIndex:UINT;
	UnsubscribeLastHighest : UINT := 16#FFFF;
	SubscribeLastHighest : UINT := 16#FFFF;
//	PublishLastHighest : UINT := 16#FFFF;
//	PubrelLastHighest : UINT := 16#FFFF;
	ReceivePaketID:WORD;
	ReceivePakteType:BYTE;
	TempSlotsWorking:UINT;
	
END_VAR
VAR CONSTANT
	
	
END_VAR
(*need a token for coordinate send of pakets....
prio for Awnser and repeat pakets bevor new publish
dont use token, just send paket with next publish index*)
//get paket id
ReceivePaketID := DWORD_TO_WORD(OSCAT_BASIC.DWORD_OF_BYTE(B3:= 0, B2:= 0, B1:= COM.R_BUF.BUFFER[2], B0:= COM.R_BUF.BUFFER[3]));
ReceivePakteType := COM.R_BUF.BUFFER[0] AND 16#F0; 

GVL_MQTT.ProgNum := PROG_NUM.STATE_MASHINE_OUT;
PublishSendListCount := 0;
PubrelSendListCount := 0;

TempSlotsWorking := 0;
FOR i := 0 TO MyConstants.IN_OUT_SLOTS_SIZE - 1 DO
	//do Timers...
	OutDataSlots[i].TimeOut(IN:= OutDataSlots[i].TimeOutStarted, PT:= MyConstants.REPEAT_TIMEOUT);
	CASE OutDataSlots[i].step OF
		
		STEPS_OUT.WAIT_DATA:
			OutDataSlots[i].TimeOutStarted := FALSE;
			IF NOT MQTT_IN_OUT^.InFree THEN//new Data from FBs
				MQTT_IN_OUT^.InFree := TRUE;
				OutDataSlots[i].InDataFromFb := MQTT_IN_OUT^.In;//set Data
				//Pakte id = slot + 1....
				OutDataSlots[i].InDataFromFb^.PaketId := i + 1;
				CASE OutDataSlots[i].InDataFromFb^.MessageType OF
					MESSAGETYPE.PINGREQ:
						OutDataSlots[i].step := STEPS_OUT.WAIT_PINGRESP;
						SendInfos.PingNeeded := TRUE;
						SendInfos.PingIndex := i;
						PingSlot := i;
					//we only sending one subscription per subscribe paket....
					MESSAGETYPE.SUBSCRIBE:
						//check if we have a slot free for subscription
						FOR j := 0 TO CALLBACKS_BUFFER_SIZE - 1 DO
							IF SubscribeCallbacks[j].free THEN
								OutDataSlots[i].step := STEPS_OUT.SEND_SUBSCRIBE;
								CallbacksFull := FALSE;
								EXIT;
							END_IF
						END_FOR
						IF j = CALLBACKS_BUFFER_SIZE THEN
							//no free slot
							MQTT_IN_OUT^.In^.CallbackError := TRUE;
							CallbacksFull := TRUE;
						END_IF
					MESSAGETYPE.UNSUBSCRIBE:
						OutDataSlots[i].step := STEPS_OUT.SEND_UNSUBSCRIBE;
					ELSE
						PushError(newError:= ERRORS.UNKNOWN_PAKET_IN_MQTT_IN_OUT , text:= CONCAT(STR1:= 'Type:', STR2:= TO_STRING(OutDataSlots[i].InDataFromFb^.MessageType)));
				END_CASE
				
			END_IF
		
		STEPS_OUT.WAIT_PINGRESP:
			IF OutDataSlots[i].TimeOutStarted AND OutDataSlots[i].TimeOut.Q AND NOT SendInfos.PingNeeded THEN
				//timeout, need repead
				SendInfos.PingNeeded := TRUE;
				SendInfos.PingIndex := i;
				CountRepeatedPing := CountRepeatedPing + 1; 
				CountRepeatedPingDisconnect := CountRepeatedPingDisconnect + 1;
				OutDataSlots[i].TimeOutStarted := FALSE;
			END_IF
		STEPS_OUT.SEND_UNSUBSCRIBE:
			//check if my paket ID is the lowest to send it
			IF OutDataSlots[i].InDataFromFb^.PaketId < UnsubscribeLastHighest AND NOT SendInfos.UnsubscribeNeeded THEN
				SendInfos.UnsubscribeIndex := i;
				SendInfos.UnsubscribeNeeded := TRUE;
				UnsubscribeLastHighest := OutDataSlots[i].InDataFromFb^.PaketId;
			END_IF	
		STEPS_OUT.WAIT_UNSUBACK:
			IF OutDataSlots[i].TimeOutStarted AND OutDataSlots[i].TimeOut.Q THEN
				//timeout, need repead
				OutDataSlots[i].step := STEPS_OUT.SEND_UNSUBSCRIBE;//repeat subscribe
				CountRepeatUnsubscribe := CountRepeatUnsubscribe + 1;
				OutDataSlots[i].TimeOutStarted := FALSE;
			END_IF
		STEPS_OUT.SEND_SUBSCRIBE:
			//check if my paket ID is the lowest to send it
			IF OutDataSlots[i].InDataFromFb^.PaketId < SubscribeLastHighest AND NOT SendInfos.SubscribeNeeded THEN
				SendInfos.SubscribeIndex := i;
				SendInfos.SubscribeNeeded := TRUE;
				SubscribeLastHighest := OutDataSlots[i].InDataFromFb^.PaketId;
			END_IF	
		STEPS_OUT.WAIT_SUBACK:
			IF OutDataSlots[i].TimeOutStarted AND OutDataSlots[i].TimeOut.Q THEN
				//timeout, need repead
				OutDataSlots[i].step := STEPS_OUT.SEND_SUBSCRIBE;//repeat subscribe
				CountRepeatSubscribe := CountRepeatSubscribe + 1;
				OutDataSlots[i].TimeOutStarted := FALSE;
			END_IF
			
		STEPS_OUT.SEND_PUBLSIH:
			PublishSendList[PublishSendListCount] := i;
			PublishSendListCount := PublishSendListCount + 1;
			
		STEPS_OUT.WAIT_PUBACK:
			IF OutDataSlots[i].TimeOutStarted AND OutDataSlots[i].TimeOut.Q THEN
				PushError(newError:= ERRORS.REPEAT_PUBLISH_PUBACK, text:= CONCAT(STR1 := CONCAT(STR1:= 'Slot:', STR2:= TO_STRING(i)),
							 STR2:= CONCAT(STR1:=', PAKET:', STR2:=TO_STRING(OutDataSlots[i].InDataFromFb^.PaketId ))));
				//timeout, need repead
				OutDataSlots[i].InDataFromFb^.DUP := TRUE;
				OutDataSlots[i].step := STEPS_OUT.SEND_PUBLSIH;//repeat publish
				RepeatedPublish := RepeatedPublish + 1;
				OutDataSlots[i].TimeOutStarted := FALSE;
			END_IF
			
		STEPS_OUT.WAIT_PUBREC:
			IF OutDataSlots[i].TimeOutStarted AND OutDataSlots[i].TimeOut.Q THEN
				PushError(newError:= ERRORS.REPEAT_PUBLISH_PUBREC, text:= CONCAT(STR1 := CONCAT(STR1:= 'Slot:', STR2:= TO_STRING(i)),
							 STR2:= CONCAT(STR1:=', PAKET:', STR2:=TO_STRING(OutDataSlots[i].InDataFromFb^.PaketId ))));
				//timeout, need repead
				OutDataSlots[i].InDataFromFb^.DUP := TRUE;
				OutDataSlots[i].step := STEPS_OUT.SEND_PUBLSIH;//repeat publish
				RepeatedPublish := RepeatedPublish + 1;
				OutDataSlots[i].TimeOutStarted := FALSE;
			END_IF
			
		STEPS_OUT.SEND_PUBREL:
			PubrelSendList[PubrelSendListCount] := i;
			PubrelSendListCount := PubrelSendListCount + 1;
			
		STEPS_OUT.WAIT_PUBCOMP:
			IF OutDataSlots[i].TimeOutStarted AND OutDataSlots[i].TimeOut.Q THEN
				//timeout, need repead
				OutDataSlots[i].step := STEPS_OUT.SEND_PUBREL;//repeat pubrel
				RepeatedPubrel := RepeatedPubrel + 1;
				OutDataSlots[i].TimeOutStarted := FALSE;
				OutDataSlots[i].PUBRELRepeatCounter := OutDataSlots[i].PUBRELRepeatCounter + 1;
				IF OutDataSlots[i].PUBRELRepeatCounter >= MyConstants.MAX_PUBREL_REPEATS THEN
					OutDataSlots[i].PUBRELRepeatCounter := 0;
					//resend publish
					OutDataSlots[i].step := STEPS_OUT.SEND_PUBLSIH;
					OutDataSlots[i].InDataFromFb^.DUP := TRUE;
					RepeatedPublishsAfterPubrel := RepeatedPublishsAfterPubrel + 1;
					PushError(newError:= ERRORS.REPEAT_PUBLISH_PUBCOMP, text:= CONCAT(STR1 := CONCAT(STR1:= 'Slot:', STR2:= TO_STRING(i)),
							 STR2:= CONCAT(STR1:=', PAKET:', STR2:=TO_STRING(OutDataSlots[i].InDataFromFb^.PaketId ))));
				ELSE
					PushError(newError:= ERRORS.REPEAT_PUBREL, text:= CONCAT(STR1 := CONCAT(STR1:= 'Slot:', STR2:= TO_STRING(i)),
							 STR2:= CONCAT(STR1:=', PAKET:', STR2:=TO_STRING(OutDataSlots[i].InDataFromFb^.PaketId ))));
				END_IF
			END_IF
		IF NOT (OutDataSlots[i].step = STEPS_OUT.WAIT_DATA) THEN
			TempSlotsWorking := TempSlotsWorking + 1;
		END_IF
	END_CASE
	//make sure timer is set to 0 if timeout resetet
	OutDataSlots[i].TimeOut(IN:= OutDataSlots[i].TimeOutStarted, PT:= MyConstants.REPEAT_TIMEOUT);
END_FOR

//now sort the arrays...
IF PublishSendListCount > 1 THEN
	FOR i := 0 TO PublishSendListCount - 1 DO
		tmpLowest := 16#FFFF;
		minIndex := i;
		FOR j := i TO PublishSendListCount - 1 DO
			IF OutDataSlots[PublishSendList[j]].PUBLISHOrder < tmpLowest THEN
				minIndex := j;
				tmpLowest := OutDataSlots[PublishSendList[j]].PUBLISHOrder;
			END_IF
		END_FOR
		IF minIndex <> i THEN
			//hier tauschen
			j := PublishSendList[minIndex];
			PublishSendList[minIndex] := PublishSendList[i];
			PublishSendList[i] := j;
		END_IF
	END_FOR
END_IF

IF PubrelSendListCount > 1 THEN
	FOR i := 0 TO PubrelSendListCount - 1 DO
		tmpLowest := 16#FFFF;
		minIndex := i;
		FOR j := i TO PubrelSendListCount - 1 DO
			IF OutDataSlots[PubrelSendList[j]].PUBRECOrder < tmpLowest THEN
				minIndex := j;
				tmpLowest := OutDataSlots[PubrelSendList[j]].PUBRECOrder;
			END_IF
		END_FOR
		IF minIndex <> i THEN
			//hier tauschen
			j := PubrelSendList[minIndex];
			PubrelSendList[minIndex] := PubrelSendList[i];
			PubrelSendList[i] := j;
		END_IF
	END_FOR
END_IF

//Hamdel PubrelOrderIndexCounter
IF PubrelOrderIndexCounter > MyConstants.REORDER_VALUE THEN 
	IF MQTT_IN_OUT^.putReordersInHistory THEN
		PushError(newError:= ERRORS.REORDER_PUBREC , text:= '');
	END_IF
	//do it brute force, just sub 20000 to every value...
	FOR i := 0 TO MyConstants.IN_OUT_SLOTS_SIZE - 1 DO
		OutDataSlots[i].PUBRECOrder := OutDataSlots[i].PUBRECOrder - MyConstants.SUBSTRACTION_VALUE;
	END_FOR
	PubrelOrderIndexCounter := MyConstants.REORDER_VALUE - MyConstants.SUBSTRACTION_VALUE + 1;
END_IF
//Hamdel PublishOrderIndexCounter
IF OutgoingPublishOrderIndexCounter > MyConstants.REORDER_VALUE THEN
	IF MQTT_IN_OUT^.putReordersInHistory THEN 
		PushError(newError:= ERRORS.REORDER_PUBLISH_OUTGOING, text:= '');
	END_IF
	//do it brute force, just sub 20000 to every value...
	FOR i := 0 TO MyConstants.IN_OUT_SLOTS_SIZE - 1 DO
		OutDataSlots[i].PUBLISHOrder := OutDataSlots[i].PUBLISHOrder - MyConstants.SUBSTRACTION_VALUE;
	END_FOR
	OutgoingPublishOrderIndexCounter := MyConstants.REORDER_VALUE - MyConstants.SUBSTRACTION_VALUE + 1;
END_IF

OutSlotsWorking := TempSlotsWorking;
END_METHOD

METHOD StateMashineIn
VAR_INPUT
	MQTT_IN_OUT : POINTER TO MQTT_IN_OUT;
END_VAR
VAR
	
	i: UINT;
	j: UINT;
	TempSlotsWorking:UINT;
	tmpLowest:UINT;
	minIndex: UINT;
END_VAR

GVL_MQTT.ProgNum := PROG_NUM.STATE_MASHINE_IN;
//Handle State Mashines
PubackSendListCount := 0;
PubrecSendListCount := 0;
PubcompSendListCount := 0;
TempSlotsWorking := 0;
FOR i := 0 TO MyConstants.IN_OUT_SLOTS_SIZE - 1 DO
	//do Timers...
	InDataSlots[i].TimeOut(IN:= InDataSlots[i].TimeOutStarted, PT:= MyConstants.REPEAT_TIMEOUT);
	IF NOT (InDataSlots[i].step = STEPS_IN.WAIT_DATA) THEN
		TempSlotsWorking := TempSlotsWorking + 1;
	END_IF  
	CASE InDataSlots[i].step OF
		STEPS_IN.WAIT_DATA:;
		STEPS_IN.WAIT_PUBREL:
		IF InDataSlots[i].TimeOut.Q THEN
			InDataSlots[i].step := STEPS_IN.SEND_PUBREC;
			InDataSlots[i].TimeOutStarted := FALSE;
			CountRepeatetPubrec := CountRepeatetPubrec + 1;
			PUBREC_ERROR_ID_BUFFER[PUBREC_ERROR_INDEX] := InDataSlots[i].PaketID; 
			PUBREC_ERROR_INDEX := PUBREC_ERROR_INDEX + 1;
			InDataSlots[i].CountPubrecRepeat := InDataSlots[i].CountPubrecRepeat + 1;
				
			IF InDataSlots[i].CountPubrecRepeat > COUNT_MAX_PUBREC_REPEAT_TO_DISCHARGE THEN
				InDataSlots[i].CountPubrecRepeat := 0;
				InDataSlots[i].step := STEPS_IN.WAIT_DATA;
				PushError(newError:= ERRORS.PUBREC_DISCHARGE, text:= CONCAT(STR1 := CONCAT(STR1:= 'Slot:', STR2:= TO_STRING(i)),
							 STR2:= CONCAT(STR1:=', PAKET:', STR2:=TO_STRING(InDataSlots[i].PaketID))));
			
			ELSE
				PushError(newError:= ERRORS.REPEAT_PUBREC, text:= CONCAT(STR1 := CONCAT(STR1:= 'Slot:', STR2:= TO_STRING(i)),
							 STR2:= CONCAT(STR1:=', PAKET:', STR2:=TO_STRING(InDataSlots[i].PaketID))));
			
			END_IF
			IF PUBREC_ERROR_INDEX >= PUBREC_ERROR_ID_BUFFER_SIZE THEN
				PUBREC_ERROR_INDEX := 0;
			END_IF
		END_IF
		STEPS_IN.SEND_PUBACK:
			PubackSendList[PubackSendListCount] := i;
			PubackSendListCount := PubackSendListCount + 1;
			
		STEPS_IN.SEND_PUBREC:
			PubrecSendList[PubrecSendListCount] := i;
			PubrecSendListCount := PubrecSendListCount + 1;
		
		STEPS_IN.SEND_PUBCOMP:
			PubcompSendList[PubcompSendListCount] := i;
			PubcompSendListCount := PubcompSendListCount + 1;
		
	END_CASE
	//make sure timer is set to 0 if timeout resetet
	InDataSlots[i].TimeOut(IN:= InDataSlots[i].TimeOutStarted, PT:= MyConstants.REPEAT_TIMEOUT);
END_FOR


//now sort the arrays...
IF PubackSendListCount > 1 THEN
	FOR i := 0 TO PubackSendListCount - 1 DO
		tmpLowest := 16#FFFF;
		minIndex := i;
		FOR j := i TO PubackSendListCount - 1 DO
			IF InDataSlots[PubackSendList[j]].PUBLISHOrder < tmpLowest THEN
				minIndex := j;
				tmpLowest := InDataSlots[PubackSendList[j]].PUBLISHOrder;
			END_IF
		END_FOR
		IF minIndex <> i THEN
			//hier tauschen
			j := PubackSendList[minIndex];
			PubackSendList[minIndex] := PubackSendList[i];
			PubackSendList[i] := j;
		END_IF
	END_FOR
END_IF

IF PubrecSendListCount > 1 THEN
	FOR i := 0 TO PubrecSendListCount - 1 DO
		tmpLowest := 16#FFFF;
		minIndex := i;
		FOR j := i TO PubrecSendListCount - 1 DO
			IF InDataSlots[PubrecSendList[j]].PUBLISHOrder < tmpLowest THEN
				minIndex := j;
				tmpLowest := InDataSlots[PubrecSendList[j]].PUBLISHOrder;
			END_IF
		END_FOR
		IF minIndex <> i THEN
			//hier tauschen
			j := PubrecSendList[minIndex];
			PubrecSendList[minIndex] := PubrecSendList[i];
			PubrecSendList[i] := j;
		END_IF
	END_FOR
END_IF


IF PubcompSendListCount > 1 THEN
	FOR i := 0 TO PubcompSendListCount - 1 DO
		tmpLowest := 16#FFFF;
		minIndex := i;
		FOR j := i TO PubcompSendListCount - 1 DO
			IF InDataSlots[PubcompSendList[j]].PUBCOMPOrder < tmpLowest THEN
				minIndex := j;
				tmpLowest := InDataSlots[PubcompSendList[j]].PUBCOMPOrder;
			END_IF
		END_FOR
		IF minIndex <> i THEN
			//hier tauschen
			j := PubcompSendList[minIndex];
			PubcompSendList[minIndex] := PubcompSendList[i];
			PubcompSendList[i] := j;
		END_IF
	END_FOR
END_IF
//Hamdel PublishOrderIndexCounter
IF IncomingPublishOrderIndexCounter > MyConstants.REORDER_VALUE THEN 
	IF MQTT_IN_OUT^.putReordersInHistory THEN
		PushError(newError:= ERRORS.REODER_PUBLISH_INCOMMING , text:= '');
	END_IF		
	//do it brute force, just sub 20000 to every value...
	FOR i := 0 TO MyConstants.IN_OUT_SLOTS_SIZE - 1 DO
		InDataSlots[i].PUBLISHOrder := InDataSlots[i].PUBLISHOrder - MyConstants.SUBSTRACTION_VALUE;
	END_FOR
	IncomingPublishOrderIndexCounter := MyConstants.REORDER_VALUE - MyConstants.SUBSTRACTION_VALUE + 1;
END_IF

//Hamdel PublishOrderIndexCounter
IF PubcompOrderIndexCounter > MyConstants.REORDER_VALUE THEN
	IF MQTT_IN_OUT^.putReordersInHistory THEN 
		PushError(newError:= ERRORS.REORDER_PUBCOMP, text:= '');
	END_IF
	//do it brute force, just sub 20000 to every value...
	FOR i := 0 TO MyConstants.IN_OUT_SLOTS_SIZE - 1 DO
		InDataSlots[i].PUBCOMPOrder := InDataSlots[i].PUBCOMPOrder - MyConstants.SUBSTRACTION_VALUE;
	END_FOR
	PubcompOrderIndexCounter := MyConstants.REORDER_VALUE - MyConstants.SUBSTRACTION_VALUE + 1;
END_IF

InSlotsWorking := TempSlotsWorking;
END_METHOD

METHOD BuildPublishPaket : BOOL
VAR_INPUT
	PaketData:POINTER TO PAKET_DATA;
	//start: BOOL;

END_VAR
VAR
	idx:UINT;
	
END_VAR
(*now change to realy big topics and payloads, do that to big topics and payloads transmitted splitted*)

BuildPublishPaket := FALSE;
IF StepBuildPublish = 0 THEN
	StepBuildPublish := 10; 
END_IF

idx := COM.S_BUF.SIZE;
//check if buffer is big enought for control, remainig length, topic size....
IF StepBuildPublish = 10 THEN

	IF (6 + COM.S_BUF.SIZE)
		 > TRANSMIT_BUFFER_SIZE THEN//only check if header fits into buffer...
		 CountCantSendPublishBufferToFull := CountCantSendPublishBufferToFull + 1;
		RETURN;	
	END_IF
	COM.S_BUF.BUFFER[idx] := MESSAGETYPE.PUBLISH;//set type
	IF PaketData^.DUP THEN//insert DUP bit
		COM.S_BUF.BUFFER[idx] := COM.S_BUF.BUFFER[idx] OR 2#1000;
	END_IF 
	COM.S_BUF.BUFFER[idx] := COM.S_BUF.BUFFER[idx] OR SHL(PaketData^.MessageQoS,1);
	IF PaketData^.MessageRetain THEN
		COM.S_BUF.BUFFER[idx] := COM.S_BUF.BUFFER[idx] OR 2#1;
	END_IF
	//do remainig lenght... 

	idx := idx + 2 + DoRemainingLengthBevor(buffer:= ADR(COM.S_BUF.BUFFER[idx]), SizeTopic:= PaketData^.MqttTopicLength, SizePayload:= PaketData^.MqttPayloadLength, InQoS:= PaketData^.MessageQoS);

	StepBuildPublish := 20;
END_IF

IF StepBuildPublish = 20 THEN
	GVL_MQTT.ProgNum := PROG_NUM.SendOutDataInsertTopic;
	//insert topic
	InsertSplitTopic(
		topic:= PaketData^.MqttTopic, 
		len:= PaketData^.MqttTopicLength, 
		buff:= ADR(COM.S_BUF.BUFFER), 
		pos:= idx, 
		size:= NETWORK_BUFFER_LONG_SIZE);
	CASE InsertSplitTopic.state OF
		INSERT_SPLIT_RETURN.INSERT_DONE:
			StepBuildPublish := 30;
		INSERT_SPLIT_RETURN.INSERT_ERROR:
			StepBuildPublish := 0;
			InsertSplitTopic.reset();
			RETURN;
		INSERT_SPLIT_RETURN.INSERT_PENDING:
			//here do nothing, just wait
		ELSE
			InsertSplitTopic.reset();
			StepBuildPublish := 0;
			RETURN;
	END_CASE
	idx := InsertSplitTopic.new_pos;
END_IF
IF StepBuildPublish = 30 THEN
	IF PaketData^.MessageQoS > 0 THEN//QoS is more then 0
		IF (2 + idx)//insert paket identifier
		 < TRANSMIT_BUFFER_SIZE THEN//enough space for identifier?
			COM.S_BUF.BUFFER[idx] := OSCAT_BASIC.BYTE_OF_DWORD(in:= PaketData^.PaketId, N:= 1);
			idx := idx + 1;
			COM.S_BUF.BUFFER[idx] := OSCAT_BASIC.BYTE_OF_DWORD(in:= PaketData^.PaketId, N:= 0);
			idx := idx + 1;
			StepBuildPublish := 40;
		END_IF
	ELSE
		StepBuildPublish := 40;
		MqttsDoneIo := MqttsDoneIo + 1;
	END_IF
END_IF

IF StepBuildPublish = 40 THEN
	GVL_MQTT.ProgNum := PROG_NUM.SendOutDataInsertPayload;
	//now insert payload
	IF PaketData^.MqttPayloadLength > 0 THEN
		//insert payload
		InsertSplitPayload(
			payload:= PaketData^.MqttPayload, 
			len:= PaketData^.MqttPayloadLength, 
			buff:= ADR(COM.S_BUF.BUFFER), 
			pos:= idx, 
			size:= NETWORK_BUFFER_LONG_SIZE);
		CASE InsertSplitPayload.state OF
			INSERT_SPLIT_RETURN.INSERT_DONE:
				StepBuildPublish := 0;
				BuildPublishPaket := TRUE;
			INSERT_SPLIT_RETURN.INSERT_ERROR:
				StepBuildPublish := 0;
				InsertSplitPayload.reset();
				RETURN;
			INSERT_SPLIT_RETURN.INSERT_PENDING:
				//here do nothing, just wait
				//or handle timeout....
			ELSE
				InsertSplitPayload.reset();
				StepBuildPublish := 0;
				RETURN;
		END_CASE
		idx := InsertSplitPayload.new_pos;
	ELSE
		StepBuildPublish := 0;
		BuildPublishPaket := TRUE;
	END_IF
END_IF
COM.S_BUF.SIZE := idx;
END_METHOD

METHOD MoveBufferForSplitPaket
VAR_INPUT
	idx:UINT;
END_VAR
VAR
	BytesToMove : UINT;
END_VAR
GVL_MQTT.ProgNum := PROG_NUM.MoveBuffer;
BytesToMove := COM.R_BUF.SIZE - idx;
CountBufferMoves := CountBufferMoves + 1;
MEM.MemMove(pSource:= ADR(com.R_BUF.BUFFER[idx]), pDestination:= ADR(com.R_BUF.BUFFER), uiNumberOfBytes:= BytesToMove);
COM.R_BUF.SIZE := BytesToMove;//manipulate size....
END_METHOD

METHOD BuildSubscribePaket : BOOL
VAR_INPUT
	PaketData:POINTER TO PAKET_DATA;
END_VAR
VAR
	idx:UINT;
	
END_VAR
BuildSubscribePaket := FALSE;
IF  StepBuildSubscribe = 0 THEN
	StepBuildSubscribe := 10;
END_IF

idx := COM.S_BUF.SIZE;
IF StepBuildSubscribe = 10 THEN
	IF (6 + COM.S_BUF.SIZE)
	 > TRANSMIT_BUFFER_SIZE THEN//only check if header fits into buffer...
		 RETURN;
	END_IF
	idx := COM.S_BUF.SIZE;
	COM.S_BUF.BUFFER[idx] := MESSAGETYPE.SUBSCRIBE OR 2#10;//set type, for 2#10 see subscribe doku
	idx := idx + 2 + DoRemainingLengthBevor(buffer:= ADR(COM.S_BUF.BUFFER[idx]), SizeTopic:= PaketData^.MqttTopicLength, SizePayload:= 1, InQoS:= QoS.AtLeastOnce);
	COM.S_BUF.BUFFER[idx] := OSCAT_BASIC.BYTE_OF_DWORD(in:= PaketData^.PaketId, N:= 1);
	idx := idx + 1;
	COM.S_BUF.BUFFER[idx] := OSCAT_BASIC.BYTE_OF_DWORD(in:= PaketData^.PaketId, N:= 0);
	idx := idx + 1;
	StepBuildSubscribe := 20;
END_IF


IF StepBuildSubscribe = 20 THEN
	//insert topic
	InsertSplitTopic(
		topic:= PaketData^.MqttTopic, 
		len:= PaketData^.MqttTopicLength, 
		buff:= ADR(COM.S_BUF.BUFFER), 
		pos:= idx, 
		size:= NETWORK_BUFFER_LONG_SIZE);
	CASE InsertSplitTopic.state OF
		INSERT_SPLIT_RETURN.INSERT_DONE:
			StepBuildSubscribe := 30;
		INSERT_SPLIT_RETURN.INSERT_ERROR:
			StepBuildSubscribe := 0;
			InsertSplitTopic.reset();
			RETURN;
		INSERT_SPLIT_RETURN.INSERT_PENDING:
			//here do nothing, just wait
		ELSE
			InsertSplitTopic.reset();
			StepBuildSubscribe := 0;
			RETURN;
	END_CASE
	idx := InsertSplitTopic.new_pos;
END_IF

IF StepBuildSubscribe = 30 THEN

	IF (1 + idx)
	 > TRANSMIT_BUFFER_SIZE THEN//only check if qos fits into buffer...
		 RETURN;
	 END_IF
	//insert QoS
	COM.S_BUF.BUFFER[idx] := PaketData^.MessageQoS;
	idx := idx + 1;
	StepBuildSubscribe := 0;
	BuildSubscribePaket := TRUE;
END_IF

COM.S_BUF.SIZE := idx;
END_METHOD

METHOD BuildUnsubscribePaket : BOOL
VAR_INPUT
	PaketData:POINTER TO PAKET_DATA;
END_VAR
VAR
	idx:UINT;
END_VAR
BuildUnsubscribePaket := FALSE;

IF  StepBuildUnsubscribe = 0 THEN
	StepBuildUnsubscribe := 10;
END_IF

idx := COM.S_BUF.SIZE;
IF StepBuildUnsubscribe = 10 THEN
	IF (6 + COM.S_BUF.SIZE)
	 > TRANSMIT_BUFFER_SIZE THEN//only check if header fits into buffer...
		 RETURN;
	END_IF
	idx := COM.S_BUF.SIZE;
	COM.S_BUF.BUFFER[idx] := MESSAGETYPE.UNSUBSCRIBE OR 2#10;//set type, for 2#10 see subscribe doku
	idx := idx + 2 + DoRemainingLengthBevor(buffer:= ADR(COM.S_BUF.BUFFER[idx]), SizeTopic:= PaketData^.MqttTopicLength, SizePayload:= 0, InQoS:= QoS.AtLeastOnce);
	COM.S_BUF.BUFFER[idx] := OSCAT_BASIC.BYTE_OF_DWORD(in:= PaketData^.PaketId, N:= 1);
	idx := idx + 1;
	COM.S_BUF.BUFFER[idx] := OSCAT_BASIC.BYTE_OF_DWORD(in:= PaketData^.PaketId, N:= 0);
	idx := idx + 1;
	StepBuildUnsubscribe := 20;
END_IF


IF StepBuildUnsubscribe = 20 THEN
	//insert topic
	InsertSplitTopic(
		topic:= PaketData^.MqttTopic, 
		len:= PaketData^.MqttTopicLength, 
		buff:= ADR(COM.S_BUF.BUFFER), 
		pos:= idx, 
		size:= NETWORK_BUFFER_LONG_SIZE);
	CASE InsertSplitTopic.state OF
		INSERT_SPLIT_RETURN.INSERT_DONE:
			StepBuildUnsubscribe := 0;
			BuildUnsubscribePaket := TRUE;
		INSERT_SPLIT_RETURN.INSERT_ERROR:
			StepBuildUnsubscribe := 0;
			InsertSplitTopic.reset();
			RETURN;
		INSERT_SPLIT_RETURN.INSERT_PENDING:
			//here do nothing, just wait
		ELSE
			InsertSplitTopic.reset();
			StepBuildUnsubscribe := 0;
			RETURN;
	END_CASE
	idx := InsertSplitTopic.new_pos;
END_IF

COM.S_BUF.SIZE := idx;
END_METHOD

METHOD SendOutData
VAR_INPUT
	//StepData:POINTER TO MQTT_OUT_DATA;
	MQTT_IN_OUT : POINTER TO MQTT_IN_OUT;
END_VAR
VAR
	SomethingIsBlocking: BOOL;
	i:UINT;
END_VAR
IF NOT SendFree THEN RETURN; END_IF
GVL_MQTT.ProgNum := PROG_NUM.SendOutData;

SomethingIsBlocking := SendInfos.PublishBlocking OR SendInfos.SubscribeBlocking OR SendInfos.UnsubscribeBlocking;

//Prio for Timeout Paket
IF  NOT (COM.S_BUF.SIZE + SIZE_PINGREQ > TRANSMIT_BUFFER_SIZE) AND SendInfos.PingNeeded AND NOT SomethingIsBlocking THEN
	SendInfos.PingNeeded := FALSE;
	COM.S_BUF.BUFFER[COM.S_BUF.SIZE] := MESSAGETYPE.PINGREQ;
	COM.S_BUF.BUFFER[COM.S_BUF.SIZE + 1] := 0;//no more length 	
	COM.S_BUF.SIZE := COM.S_BUF.SIZE + SIZE_PINGREQ;//small ping paket
	OutDataSlots[SendInfos.PingIndex].TimeOutStarted := TRUE;//start Timeout
END_IF
IF NOT COM.S_BUF.SIZE = 0 THEN 
	CountOutSendNotFree := CountOutSendNotFree + 1;
END_IF
//next Prio send Pubrel 
IF PubrelSendListCount > 0 AND NOT SomethingIsBlocking THEN
	FOR i := 0 TO PubrelSendListCount - 1 DO
		IF NOT (COM.S_BUF.SIZE + SIZE_PUBREL > TRANSMIT_BUFFER_SIZE) THEN
			COM.S_BUF.BUFFER[COM.S_BUF.SIZE] := MESSAGETYPE.PUBREL OR 2#10;//set type and Reserved bits
			COM.S_BUF.BUFFER[COM.S_BUF.SIZE + 1] := 2;
			COM.S_BUF.BUFFER[COM.S_BUF.SIZE + 2] := OSCAT_BASIC.BYTE_OF_DWORD(in:= OutDataSlots[PubrelSendList[i]].InDataFromFb^.PaketId, N:= 1);
			COM.S_BUF.BUFFER[COM.S_BUF.SIZE + 3] := OSCAT_BASIC.BYTE_OF_DWORD(in:= OutDataSlots[PubrelSendList[i]].InDataFromFb^.PaketId, N:= 0);
			COM.S_BUF.SIZE := COM.S_BUF.SIZE + SIZE_PUBREL;
			OutDataSlots[PubrelSendList[i]].step := STEPS_OUT.WAIT_PUBCOMP;
			OutDataSlots[PubrelSendList[i]].TimeOutStarted := TRUE;//start Timeout			
		ELSE
			EXIT;
		END_IF 
	END_FOR
END_IF

//send Unsubscribe
IF SendInfos.UnsubscribeNeeded AND (NOT SomethingIsBlocking OR SendInfos.UnsubscribeBlocking) THEN
	IF NOT BuildUnsubscribePaket(PaketData:= OutDataSlots[SendInfos.UnsubscribeIndex].InDataFromFb) THEN
		SendInfos.UnsubscribeBlocking := TRUE;
	ELSE
		SendInfos.UnsubscribeBlocking := FALSE;
		SendInfos.UnsubscribeNeeded := FALSE;
		OutDataSlots[SendInfos.UnsubscribeIndex].TimeOutStarted := TRUE;
		OutDataSlots[SendInfos.UnsubscribeIndex].step := STEPS_OUT.WAIT_UNSUBACK;
	END_IF
END_IF

//send Subscribe
IF SendInfos.SubscribeNeeded AND (NOT SomethingIsBlocking OR SendInfos.SubscribeBlocking) THEN
	IF NOT BuildSubscribePaket(PaketData:= OutDataSlots[SendInfos.SubscribeIndex].InDataFromFb) THEN
		SendInfos.SubscribeBlocking := TRUE;
	ELSE
		SendInfos.SubscribeBlocking := FALSE;
		SendInfos.SubscribeNeeded := FALSE;
		OutDataSlots[SendInfos.SubscribeIndex].TimeOutStarted := TRUE;
		OutDataSlots[SendInfos.SubscribeIndex].step := STEPS_OUT.WAIT_SUBACK;
	END_IF
END_IF
//send pending Publish 
IF SendInfos.PublishBlocking THEN
	IF BuildPublishPaket(PaketData:= OutDataSlots[SendInfos.PublishBlockingIndex].InDataFromFb) THEN
		SendInfos.PublishBlocking := FALSE;
		PublishSendDone(slot:=ADR(OutDataSlots[SendInfos.PublishBlockingIndex]));
	END_IF
END_IF

IF (PublishSendListCount > 0 AND NOT SomethingIsBlocking) THEN
	//handle pendig publisah packet
	//handle new publish packet
	FOR i := 0 TO PublishSendListCount - 1 DO
		IF NOT BuildPublishPaket(PaketData:= OutDataSlots[PublishSendList[i]].InDataFromFb) THEN
			SendInfos.PublishBlocking := TRUE;
			SendInfos.PublishBlockingIndex := PublishSendList[i];
			EXIT;
		ELSE 
			SendInfos.PublishBlocking := FALSE;
			PublishSendDone(slot:=ADR(OutDataSlots[PublishSendList[i]]));
		END_IF
	END_FOR
END_IF
END_METHOD

METHOD SendInData
VAR_INPUT
	MQTT_IN_OUT : POINTER TO MQTT_IN_OUT;
END_VAR
VAR
	i : UINT;
END_VAR
IF NOT SendFree THEN RETURN; END_IF

GVL_MQTT.ProgNum := PROG_NUM.SendInData;

IF NOT COM.S_BUF.SIZE = 0 THEN 
	CountInSendNotFree := CountInSendNotFree + 1;
END_IF

IF PubackSendListCount > 0 THEN
	FOR i := 0 TO PubackSendListCount - 1 DO
		IF NOT (COM.S_BUF.SIZE + SIZE_PUBACK > TRANSMIT_BUFFER_SIZE)  THEN
			COM.S_BUF.BUFFER[COM.S_BUF.SIZE] := MESSAGETYPE.PUBACK;
			COM.S_BUF.BUFFER[COM.S_BUF.SIZE + 1] := 2;//length of 2
			COM.S_BUF.BUFFER[COM.S_BUF.SIZE + 2] := OSCAT_BASIC.BYTE_OF_DWORD(in:= InDataSlots[PubackSendList[i]].PaketID, N:= 1);
			COM.S_BUF.BUFFER[COM.S_BUF.SIZE + 3] := OSCAT_BASIC.BYTE_OF_DWORD(in:= InDataSlots[PubackSendList[i]].PaketID, N:= 0);
			COM.S_BUF.SIZE := COM.S_BUF.SIZE + SIZE_PUBACK;//Paket size allways 4!
			InDataSlots[PubackSendList[i]].step := STEPS_IN.WAIT_DATA;
			MqttsDoneIo := MqttsDoneIo + 1;	
		ELSE
			EXIT;
		END_IF
	END_FOR
	
END_IF

IF PubcompSendListCount > 0 THEN
	FOR i := 0 TO PubcompSendListCount - 1 DO
		IF NOT (COM.S_BUF.SIZE + SIZE_PUBCOMP > TRANSMIT_BUFFER_SIZE) THEN	
			COM.S_BUF.BUFFER[COM.S_BUF.SIZE] := MESSAGETYPE.PUBCOMP;
			COM.S_BUF.BUFFER[COM.S_BUF.SIZE + 1] := 2;//length of 2
			COM.S_BUF.BUFFER[COM.S_BUF.SIZE + 2] := OSCAT_BASIC.BYTE_OF_DWORD(in:= InDataSlots[PubcompSendList[i]].PaketID, N:= 1);
			COM.S_BUF.BUFFER[COM.S_BUF.SIZE + 3] := OSCAT_BASIC.BYTE_OF_DWORD(in:= InDataSlots[PubcompSendList[i]].PaketID, N:= 0);
			COM.S_BUF.SIZE := COM.S_BUF.SIZE + SIZE_PUBCOMP;//Paket size allways 4!
			InDataSlots[PubcompSendList[i]].step := STEPS_IN.WAIT_DATA;
			MqttsDoneIo := MqttsDoneIo + 1;
		ELSE
			EXIT;
		END_IF
	END_FOR
END_IF

IF PubrecSendListCount > 0 THEN
	FOR i := 0 TO PubrecSendListCount - 1 DO
		IF NOT (COM.S_BUF.SIZE + SIZE_PUBREC > TRANSMIT_BUFFER_SIZE) THEN
			COM.S_BUF.BUFFER[COM.S_BUF.SIZE] := MESSAGETYPE.PUBREC;
			COM.S_BUF.BUFFER[COM.S_BUF.SIZE + 1] := 2;//length of 2
			COM.S_BUF.BUFFER[COM.S_BUF.SIZE + 2] := OSCAT_BASIC.BYTE_OF_DWORD(in:= InDataSlots[PubrecSendList[i]].PaketID, N:= 1);
			COM.S_BUF.BUFFER[COM.S_BUF.SIZE + 3] := OSCAT_BASIC.BYTE_OF_DWORD(in:= InDataSlots[PubrecSendList[i]].PaketID, N:= 0);
			COM.S_BUF.SIZE := COM.S_BUF.SIZE + SIZE_PUBREC;//Paket size allways 4!
			InDataSlots[PubrecSendList[i]].step := STEPS_IN.WAIT_PUBREL;
			InDataSlots[PubrecSendList[i]].TimeOutStarted := TRUE;
		ELSE
			EXIT;
		END_IF
	END_FOR
END_IF
END_METHOD

METHOD ParseIncoming
VAR_INPUT
	MQTT_IN_OUT : POINTER TO MQTT_IN_OUT;
END_VAR
VAR
	I:UINT;
	j:UINT;
	idx:UINT := 0;
	//idxFromParsePublish:UINT := 0;
	ReceivePakteType:MESSAGETYPE;
	ReceivePaketID:WORD;
	BufferMoveDone:BOOL;
	PaketFound: BOOL;

END_VAR
GVL_MQTT.ProgNum := PROG_NUM.ParseIncomming;
IF COM.R_BUF.SIZE > 0 THEN
	REPEAT
		
		PaketFound := FALSE;
		HelperLastPaktetForUnkownPaket := ReceivePakteType;
		ReceivePakteType := COM.R_BUF.BUFFER[idx] AND 16#F0;
		 
		CASE ReceivePakteType OF
			MESSAGETYPE.PUBLISH:
			//new way, move every publish to receive buffer, and then pars it.
			//outgoing payload pointer is then set to start of payload in the buffer....
				BufferMoveDone := CheckLenghtBuffer(IdxIn:= idx);
				IF NOT BufferMoveDone THEN
					
					idx := ParseIncomingPublish(MQTT_IN_OUT:= MQTT_IN_OUT, idx:= idx,
											BufferIn:= ADR(COM.R_BUF.BUFFER), BufferSize:= COM.R_BUF.SIZE,
											NetworkBuffer:= TRUE);

				END_IF
			MESSAGETYPE.PUBREL:
				BufferMoveDone := CheckLenghtBuffer(IdxIn:= idx);
				IF NOT BufferMoveDone THEN
					//get Paket ID
					ReceivePaketID := DWORD_TO_WORD(OSCAT_BASIC.DWORD_OF_BYTE(B3:= 0, B2:= 0, 
						B1:= COM.R_BUF.BUFFER[idx + 2],
						B0:= COM.R_BUF.BUFFER[idx + 3]));
					//find Paket
					FOR i := 0 TO MyConstants.IN_OUT_SLOTS_SIZE - 1 DO
						IF InDataSlots[i].PaketID = ReceivePaketID THEN
							InDataSlots[i].step := STEPS_IN.SEND_PUBCOMP;
							InDataSlots[i].TimeOutStarted := FALSE;
							PubcompOrderIndexCounter := PubcompOrderIndexCounter;
							InDataSlots[i].PUBCOMPOrder := PubcompOrderIndexCounter;
							PaketFound := TRUE;
							EXIT;
						END_IF
						//
					END_FOR
					IF NOT PaketFound THEN
						CountReceivePubrelUnknown := CountReceivePubrelUnknown + 1;
					END_IF
					idx := idx + SIZE_PUBREL;
				END_IF
			MESSAGETYPE.PINGRESP:
				ResetPingTime();
				PingRequestet := FALSE;
				OutDataSlots[PingSlot].step := STEPS_OUT.WAIT_DATA;//can get new data
				OutDataSlots[PingSlot].TimeOutStarted := FALSE;
				idx := idx + SIZE_PINGRESP;
				MqttsDoneIo := MqttsDoneIo + 1;
			MESSAGETYPE.UNSUBACK:
				BufferMoveDone := CheckLenghtBuffer(IdxIn:= idx);
				IF NOT BufferMoveDone THEN
					//get Paket ID
					ReceivePaketID := DWORD_TO_WORD(OSCAT_BASIC.DWORD_OF_BYTE(B3:= 0, B2:= 0, 
						B1:= COM.R_BUF.BUFFER[idx + 2],
						B0:= COM.R_BUF.BUFFER[idx + 3]));
					//find Paket
					FOR i := 0 TO MyConstants.IN_OUT_SLOTS_SIZE - 1 DO
						IF OutDataSlots[i].step = STEPS_OUT.WAIT_UNSUBACK THEN //make sure pointer is vailid
							IF OutDataSlots[i].InDataFromFb^.PaketId = ReceivePaketID THEN
								OutDataSlots[i].InDataFromFb^.SendSucsess := TRUE;
								OutDataSlots[i].step := STEPS_OUT.WAIT_DATA;//can get new data
								OutDataSlots[i].TimeOutStarted := FALSE;
								MqttsDoneIo := MqttsDoneIo + 1;
								PaketFound := TRUE;
								//now kick of Callback
								FOR j := 0 TO CALLBACKS_BUFFER_SIZE - 1 DO
									IF SubscribeCallbacks[j].Callback = OutDataSlots[i].InDataFromFb^.Callback  THEN
										//callback found, now kill it...
										SubscribeCallbacks[j].free := TRUE;
										SubscribeCallbacks[j].Callback := 0;
										EXIT;
									END_IF
								END_FOR
								EXIT;
							END_IF
						END_IF
						//
					END_FOR
					IF NOT PaketFound THEN
						CountReceiveUnsubackUnknown := CountReceiveUnsubackUnknown + 1;
					END_IF
					idx := idx + SIZE_UNSUBACK;	
				END_IF
				
			MESSAGETYPE.SUBACK:
				BufferMoveDone := CheckLenghtBuffer(IdxIn:= idx);
				IF NOT BufferMoveDone THEN
					//get Paket ID
					ReceivePaketID := DWORD_TO_WORD(OSCAT_BASIC.DWORD_OF_BYTE(B3:= 0, B2:= 0, 
						B1:= COM.R_BUF.BUFFER[idx + 2],
						B0:= COM.R_BUF.BUFFER[idx + 3]));
					//find Paket
					FOR i := 0 TO MyConstants.IN_OUT_SLOTS_SIZE - 1 DO
						IF OutDataSlots[i].step = STEPS_OUT.WAIT_SUBACK THEN //make sure pointer is vailid
							IF OutDataSlots[i].InDataFromFb^.PaketId = ReceivePaketID THEN
								OutDataSlots[i].InDataFromFb^.SendSucsess := TRUE;
								OutDataSlots[i].InDataFromFb^.SubackQoS := COM.R_BUF.BUFFER[idx + 4];
								OutDataSlots[i].step := STEPS_OUT.WAIT_DATA;//can get new data
								OutDataSlots[i].TimeOutStarted := FALSE;
								MqttsDoneIo := MqttsDoneIo + 1;
								PaketFound := TRUE;
								//now register callback:
								FOR j := 0 TO CALLBACKS_BUFFER_SIZE - 1 DO
									IF SubscribeCallbacks[j].free THEN
										SubscribeCallbacks[j].free := FALSE;
										SubscribeCallbacks[j].Callback := OutDataSlots[i].InDataFromFb^.Callback;
 										SubscribeCallbacks[j].SplitTopic := OutDataSlots[i].InDataFromFb^.SplitTopic;
										SubscribeCallbacks[j].ExpectingString := OutDataSlots[i].InDataFromFb^.ExpectingString;
										EXIT;
									END_IF
								END_FOR
								IF j = CALLBACKS_BUFFER_SIZE THEN
									//no callback slot free
									OutDataSlots[i].InDataFromFb^.CallbackError := TRUE;
								END_IF
								EXIT;
							END_IF
						END_IF
						//
					END_FOR
					IF NOT PaketFound THEN
						CountReceiveSubackUnknown := CountReceiveSubackUnknown + 1;
					END_IF
					idx := idx + SIZE_SUBACK;//only one QoS response expected
				END_IF
			MESSAGETYPE.PUBACK:
				BufferMoveDone := CheckLenghtBuffer(IdxIn:= idx);
				IF NOT BufferMoveDone THEN
					//get Paket ID
					ReceivePaketID := DWORD_TO_WORD(OSCAT_BASIC.DWORD_OF_BYTE(B3:= 0, B2:= 0, 
						B1:= COM.R_BUF.BUFFER[idx + 2],
						B0:= COM.R_BUF.BUFFER[idx + 3]));
					//find Paket
					FOR i := 0 TO MyConstants.IN_OUT_SLOTS_SIZE - 1 DO
						IF OutDataSlots[i].step = STEPS_OUT.WAIT_PUBACK THEN //make sure pointer is vailid
							IF OutDataSlots[i].InDataFromFb^.PaketId = ReceivePaketID THEN
								OutDataSlots[i].InDataFromFb^.SendSucsess := TRUE;
								OutDataSlots[i].step := STEPS_OUT.WAIT_DATA;//can get new data
								OutDataSlots[i].TimeOutStarted := FALSE;
								MqttsDoneIo := MqttsDoneIo + 1;
								Publishsunacknowledged := Publishsunacknowledged - 1;
								PaketFound := TRUE; 
								EXIT;
							END_IF
						END_IF
						//
					END_FOR
					IF NOT PaketFound THEN
						CountReceivePubackUnknown := CountReceivePubackUnknown + 1;
					END_IF
					idx := idx + SIZE_PUBACK;
				END_IF
			MESSAGETYPE.PUBREC:
				BufferMoveDone := CheckLenghtBuffer(IdxIn:= idx);
				IF NOT BufferMoveDone THEN
					//get Paket ID
					ReceivePaketID := DWORD_TO_WORD(OSCAT_BASIC.DWORD_OF_BYTE(B3:= 0, B2:= 0, 
						B1:= COM.R_BUF.BUFFER[idx + 2],
						B0:= COM.R_BUF.BUFFER[idx + 3]));
					//find Paket
					FOR i := 0 TO MyConstants.IN_OUT_SLOTS_SIZE - 1 DO
						IF OutDataSlots[i].step = STEPS_OUT.WAIT_PUBREC THEN //make sure pointer is vailid
							IF OutDataSlots[i].InDataFromFb^.PaketId = ReceivePaketID THEN
								IF NOT OutDataSlots[i].InDataFromFb^.DUP THEN
									//increase only at first handle 
									PubrelOrderIndexCounter := PubrelOrderIndexCounter + 1;
									OutDataSlots[i].PUBRECOrder := PubrelOrderIndexCounter;
								END_IF
								OutDataSlots[i].step := STEPS_OUT.SEND_PUBREL;
								OutDataSlots[i].TimeOutStarted := FALSE;
								PaketFound := TRUE; 
								EXIT;
							END_IF
						END_IF
						//
					END_FOR
					IF NOT PaketFound THEN
						CountReceivePubrecUnknown := CountReceivePubrecUnknown + 1;
					END_IF
					idx := idx + SIZE_PUBREC;
				END_IF
			MESSAGETYPE.PUBCOMP:
				BufferMoveDone := CheckLenghtBuffer(IdxIn:= idx);
				IF NOT BufferMoveDone THEN
					//get Paket ID
					ReceivePaketID := DWORD_TO_WORD(OSCAT_BASIC.DWORD_OF_BYTE(B3:= 0, B2:= 0, 
						B1:= COM.R_BUF.BUFFER[idx + 2],
						B0:= COM.R_BUF.BUFFER[idx + 3]));
					//find Paket
					FOR i := 0 TO MyConstants.IN_OUT_SLOTS_SIZE - 1 DO
						IF OutDataSlots[i].step = STEPS_OUT.WAIT_PUBCOMP THEN //make sure pointer is vailid
							IF OutDataSlots[i].InDataFromFb^.PaketId = ReceivePaketID THEN
								OutDataSlots[i].InDataFromFb^.SendSucsess := TRUE;
								OutDataSlots[i].step := STEPS_OUT.WAIT_DATA;//can get new data
								OutDataSlots[i].TimeOutStarted := FALSE;
								MqttsDoneIo := MqttsDoneIo + 1;
								Publishsunacknowledged := Publishsunacknowledged - 1;
								PaketFound := TRUE;
								EXIT;
							END_IF
						END_IF
						//
					END_FOR
					IF NOT PaketFound THEN
						CountReceivePubcompUnknown := CountReceivePubcompUnknown + 1;
					END_IF
					idx := idx + SIZE_PUBCOMP;			
				END_IF
			ELSE
				//unknown paket, reset buffer....
				//standard wants to disconnect....
				{info 'unkown packet, disconnect'}
				LastPaktetForUnkownPaket := HelperLastPaktetForUnkownPaket;
				COM.R_BUF.SIZE := 0;	
				//unknown paket received
				NotKnownPaket := COM.R_BUF.BUFFER[0] AND 16#F0;
				PushError(newError:= ERRORS.UNKNOWN_PAKET_RECEIVED , text:='');
				//alway reset receive!
				COM.MQTT_RCV_STATE := BYTE#0;//receive zurücksetzten
				COM.R_BUF.SIZE := 0;
				CountUnkownPaket := CountUnkownPaket + 1;	
		END_CASE
	UNTIL
		idx >= COM.R_BUF.SIZE OR BufferMoveDone
	END_REPEAT
	IF NOT BufferMoveDone THEN
		COM.R_BUF.SIZE := 0;
	END_IF
	COM.MQTT_RCV_STATE := BYTE#0;//receive zurücksetzten
	
END_IF
END_METHOD

METHOD ParseIncomingPublish :UINT
VAR_INPUT
	MQTT_IN_OUT : POINTER TO MQTT_IN_OUT;
	//pos of paket in buffer
	idx:UINT;
	//give here the buffer were the full packet is...
	BufferIn:POINTER TO BYTE;
	//works on network buffer --> need memmove in Output
	NetworkBuffer: BOOL;

	//size of buffer, bytes occupied
	BufferSize:UDINT;
END_VAR
VAR
	i:UINT;
	PaketFound: BOOL;
	PaketIndex:UINT;
	FreeSlot:UINT;
	FreeSlotFound: BOOL;
	ReceivePaketID:WORD;
	ReceiveQoSLevel:QoS;
	TopicSize:UINT;
	//Output the Data, Tru if Data can be outputted
	OutData:BOOL;
	RemainingLength:REMAINING_LENGTH_RETURN;
	PayloadPosStart:UDINT;
	TopicPosStart:UDINT;
	PayloadSize:UDINT;
	
	FollowingDataBuffer:ARRAY[0..1] OF BYTE;
	
	PayloadMoved: BOOL;

END_VAR
ParseIncomingPublish := 0;//if return is zero, buffer move has been done,
CounterPublishReceivedForMonitor := CounterPublishReceivedForMonitor + 1;
GVL_MQTT.ProgNum := PROG_NUM.ParsePublish;
//get remaining length
RemainingLength := GetRemainingLength(BufferIn, pos := idx,BuffSize := BufferSize);
TopicPosStart := RemainingLength.IndexAfterRemainingLength + 2;
ReceiveQoSLevel := SHR(BufferIn[idx] AND 2#110,1);

TopicSize := DWORD_TO_WORD(OSCAT_BASIC.DWORD_OF_BYTE(B3:= 0, B2:= 0,
						 B1:= BufferIn[RemainingLength.IndexAfterRemainingLength],
						 B0:= BufferIn[RemainingLength.IndexAfterRemainingLength+1]));
IF RemainingLength.Error THEN
	//throw away paket on length error
	COM.MQTT_RCV_STATE := BYTE#0;//receive zurücksetzten
	//need to set size to zero, so no further parsing...
	COM.R_BUF.SIZE := 0;
	CountLengthErrors := CountLengthErrors;
	//on standard i MUST diconnect!!!
	DoDisconnect := TRUE;
	PushError(newError:= ERRORS.RECEIVED_PUBLISH_REMAINING_LENGTH_ERROR, text:='');
	
	RETURN;
END_IF
//publish received, size is handleable
IF ReceiveQoSLevel = QoS.AtMostOnce THEN
	//Nothing to do, just output the Payload and Topic
	OutData := TRUE;
	PayloadSize := RemainingLength.RemainingLength - TopicSize - 2;//2 for Size Encoding
	PayloadPosStart := RemainingLength.IndexAfterRemainingLength + TopicSize + 2;//2 for Size Encoding
	CountReceivedPublishs := CountReceivedPublishs + 1;
	MqttsDoneIo := MqttsDoneIo + 1;
ELSE
	//get Paket ID
	ReceivePaketID := DWORD_TO_WORD(OSCAT_BASIC.DWORD_OF_BYTE(B3:= 0, B2:= 0, 
		B1:= BufferIn[RemainingLength.IndexAfterRemainingLength + TopicSize + 2],//+ 2 for Topic Length
		B0:= BufferIn[RemainingLength.IndexAfterRemainingLength + TopicSize + 3]));
	//2 for size of Paket identifier
	PayloadSize := RemainingLength.RemainingLength - TopicSize - 4;//2 for size of topic  and 2 for message id
	PayloadPosStart := RemainingLength.IndexAfterRemainingLength + TopicSize + 4;//2 for size of topic and 2 for message id
	
	//QoS stuff
	FOR i := 0 TO MyConstants.IN_OUT_SLOTS_SIZE - 1 DO
		IF InDataSlots[i].PaketID = ReceivePaketID AND InDataSlots[i].step <> STEPS_IN.WAIT_DATA THEN
			PaketIndex := i;
			PaketFound := TRUE;
			
		END_IF
		IF InDataSlots[i].step = STEPS_IN.WAIT_DATA AND NOT FreeSlotFound THEN
			FreeSlot := i;
			FreeSlotFound := TRUE;
		END_IF
		IF FreeSlotFound AND PaketFound THEN
			EXIT;//exit if slot and paket found
		END_IF
	END_FOR
	IF NOT PaketFound THEN
		IF FreeSlotFound THEN
			//Paket ist not to be awnserd --> first occurence
			InDataSlots[FreeSlot].CountPubrecRepeat := 0;
			InDataSlots[FreeSlot].QoS := ReceiveQoSLevel;
			InDataSlots[FreeSlot].PaketID := ReceivePaketID;
			IncomingPublishOrderIndexCounter := IncomingPublishOrderIndexCounter + 1;
			InDataSlots[FreeSlot].PUBLISHOrder := IncomingPublishOrderIndexCounter;
			OutData := TRUE;
			CountReceivedPublishs := CountReceivedPublishs + 1;
		ELSE
			//no more slots free
			{info 'no more slots free, what shall we do???'}
			//at all this is fine....
			DoDisconnect := TRUE;
			PushError(newError:= ERRORS.NO_MORE_RECEIVE_SLOTS_FREE , text:='');
			
		END_IF
	ELSE
		CountRepeatPublishReceive := CountRepeatPublishReceive + 1;
	END_IF
	CASE InDataSlots[FreeSlot].QoS OF
		QoS.AtLeastOnce:
			InDataSlots[FreeSlot].step := STEPS_IN.SEND_PUBACK;
		QoS.ExactlyOnce:
			InDataSlots[FreeSlot].step := STEPS_IN.SEND_PUBREC;
	END_CASE
END_IF

IF RemainingLength.RemainingLength > (COM_CONFIG.MaxTopicElementSize * COM_CONFIG.MaxTopicLevels + COM_CONFIG.MaxPayloadSize) OR 
	TopicSize > (COM_CONFIG.MaxTopicElementSize * COM_CONFIG.MaxTopicLevels) OR
	PayloadSize > COM_CONFIG.MaxPayloadSize THEN
	{info 'check here if to disconnect'}
	//paket to big for my Strings, but do QoS stuff!!!! no standard, standard wants disconnect!
	PushError(newError:= ERRORS.TO_BIG_PAKET , text:='');
	CountToBigTopics := CountToBigTopics  + 1;
	{info 'check if last to big topic is to saved, or just take memmove'}
	(*LastToBigTopic := OSCAT_BASIC.BUFFER_TO_STRING(PT:= ADR(BufferIn[idx]), SIZE:= BufferSize,
						START:= RemainingLength.IndexAfterRemainingLength + 2,
						STOP:= RemainingLength.IndexAfterRemainingLength + TopicSize);*)
	OutData := FALSE;//reset out Data....
END_IF


//now set idx to next packet
ParseIncomingPublish := UDINT_TO_UINT(PayloadPosStart + PayloadSize);

IF OutData THEN
		
		//new approach: in buffer for big packets we can move as we want. in network buffer, we can move topic
		//without trobble down, length information isn't needed anymore. if we move in network buffer we store 
		//the following two bytes of payload, making the output and there after we restore them.
		//this we do in buffer for big packets too, because it isn't expensive
		//but we have to be aware if the payload is near the buffer end, then we have to move it down...

		//we need to check if  
		
		//IF NOT NetworkBuffer THEN //in network buffer, we have to set an termination
		PayloadMoved := FALSE;	
		//first check if payload needs to be moved, because it is at the buffer end
		IF NetworkBuffer THEN
			IF ReceiveQoSLevel = QoS.AtMostOnce THEN//if QoS zero, we need to move, because space for packet ID is missing...
				//check which is smaller, this is to be moved....
				IF TopicSize < PayloadSize THEN
					//move Topic down
					MEM.MemMove(pSource:= ADR(BufferIn[TopicPosStart]), pDestination:= ADR(BufferIn[TopicPosStart - 1]), uiNumberOfBytes:= TopicSize);
					TopicPosStart := TopicPosStart - 1;//now topic resits one deeper
					IF LogBufferMoves THEN
						PushError(newError:= ERRORS.TOPIC_MOVED_DOWN , text:='');
					END_IF
				ELSE
					IF idx + PayloadPosStart + PayloadSize > MyConstants.NETWORK_BUFFER_LONG_SIZE THEN
						//need to move payload and topic, I'm at the top border of network buffer
						//should be very rare....
						SysMem.SysMemMove(pDest:= ADR(BufferIn[TopicPosStart - 2]), pSrc:= ADR(BufferIn[TopicPosStart]), udiCount:= TO_UDINT(TopicSize));
						SysMem.SysMemMove(pDest:= ADR(BufferIn[PayloadPosStart - 1]), pSrc:= ADR(BufferIn[PayloadPosStart]), udiCount:= TO_UDINT(PayloadSize));
						//change Topic Pointer...
						TopicPosStart := TopicPosStart - 2;
						//change Payload Pointer
						PayloadPosStart := PayloadPosStart - 1;
						IF LogBufferMoves THEN
							PushError(newError:= ERRORS.TOPIC_AND_PAYLOAD_MOVED, text:='');
						END_IF
					ELSE
						//first, save following data
						//move Payload up
						PayloadMoved := TRUE;
						FollowingDataBuffer[0] := BufferIn[PayloadPosStart + PayloadSize];
						SysMem.SysMemMove(pDest:= ADR(BufferIn[PayloadPosStart + 1]), pSrc:= ADR(BufferIn[PayloadPosStart]), udiCount:= TO_UDINT(PayloadSize));
						PayloadPosStart := PayloadPosStart + 1;//payload now resits one higher
						IF LogBufferMoves THEN
							PushError(newError:= ERRORS.PAYLOAD_MOVED_UP, text:='');
						END_IF
					END_IF
				END_IF
			END_IF
			
			//alway set termination for payload because it could be a string
			FollowingDataBuffer[1] := BufferIn[PayloadPosStart + PayloadSize]; 
			BufferIn[PayloadPosStart + PayloadSize] := 0;	
			//now set termination, if not QoS zero, overwrite PacketID
			BufferIn[TopicPosStart + TopicSize] := 0;
			//END_IF
			OutputPublish(
				PayloadSize:= PayloadSize, 
				PayloadPos:= ADR(BufferIn[PayloadPosStart]), 
				TopicSize:= TopicSize, 
				TopicPos:= ADR(BufferIn[TopicPosStart]), 
				MQTT_IN_OUT:= MQTT_IN_OUT);
			//restore data after payload
			BufferIn[PayloadPosStart + PayloadSize] := FollowingDataBuffer[1];
			//END_IF

		ELSE
			
		//here we are not in the network buffer, borders don't care and following bytes doesn't matter.
			IF ReceiveQoSLevel = QoS.AtMostOnce THEN//if QoS zero, we need to move, because space for packet ID is missing...
				//check which is smaller, this is to be moved....
				IF TopicSize < PayloadSize THEN
					//move Topic down
					MEM.MemMove(pSource:= ADR(BufferIn[TopicPosStart]), pDestination:= ADR(BufferIn[TopicPosStart - 1]), uiNumberOfBytes:= TopicSize);
					TopicPosStart := TopicPosStart - 1;//now topic resits one deeper
					IF LogBufferMoves THEN
						PushError(newError:= ERRORS.TOPIC_MOVED_DOWN_NETWORK, text:='');
					END_IF
				ELSE
					//move Payload up
					SysMem.SysMemMove(pDest:= ADR(BufferIn[PayloadPosStart + 1]), pSrc:= ADR(BufferIn[PayloadPosStart]), udiCount:= TO_UDINT(PayloadSize));
					PayloadPosStart := PayloadPosStart + 1;//payload now resits one higher
					IF LogBufferMoves THEN
						PushError(newError:= ERRORS.PAYLOAD_MOVED_UP_NETWORK, text:='');
					END_IF
				END_IF
			END_IF
			//alway set termination for payload because it could be a string
			BufferIn[PayloadPosStart + PayloadSize] := 0;	
			//now set termination, if not QoS zero, overwrite PacketID
			BufferIn[TopicPosStart + TopicSize] := 0;
			//END_IF
			OutputPublish(
				PayloadSize:= PayloadSize, 
				PayloadPos:= ADR(BufferIn[PayloadPosStart]), 
				TopicSize:= TopicSize, 
				TopicPos:= ADR(BufferIn[TopicPosStart]), 
				MQTT_IN_OUT:= MQTT_IN_OUT);
			
		END_IF
END_IF

IF PayloadMoved THEN 
	//if payload was moved, then content have to be rebuild
	BufferIn[PayloadPosStart + PayloadSize - 1] := FollowingDataBuffer[0];
END_IF
END_METHOD

METHOD CheckLenghtBuffer : BOOL 
VAR_INPUT
	IdxIn : UINT;
END_VAR
VAR
	
	ReceivePakteType: MESSAGETYPE;
	
	RemainingLength: REMAINING_LENGTH_RETURN;
	
	NeedBufferMove: BOOL;

END_VAR
ReceivePakteType := COM.R_BUF.BUFFER[IdxIn] AND 16#F0;

NeedBufferMove := FALSE;

CASE ReceivePakteType OF

	MESSAGETYPE.PUBLISH:
		IF IdxIn + 1 > COM.R_BUF.SIZE THEN//1 for min size of remaining length
			NeedBufferMove := TRUE;//maybe we at the end of the buffer, so move...
		ELSE
			//size big enough to test remaining lengt, inside testing of bytes....
			RemainingLength := GetRemainingLength(ADR(COM.R_BUF.BUFFER), pos := IdxIn, BuffSize:= COM.R_BUF.SIZE);
			//if paket to small for buffer, disconnect, remaining length is smaller then whole packet size
			IF ((TO_LINT(RemainingLength.RemainingLength) - 8 > MaxPublishPacketSize) OR RemainingLength.RemainingLength = 0) AND NOT RemainingLength.BuffToSmall THEN
				{info 'make this to a parameter to chose disconnect or discharge'}
				DoDisconnect := TRUE;
				PushError(newError:= ERRORS.RECEIVED_PUBISH_TO_BIG_FOR_BUFFER, text:='');
				CheckLenghtBuffer := TRUE;
			ELSE 
				IF RemainingLength.BuffToSmall THEN
					NeedBufferMove := TRUE;
				ELSE
					IF RemainingLength.RemainingLength < TRANSMIT_BUFFER_SIZE THEN 
						//here the packet fits into the network buffer
						IF (RemainingLength.IndexAfterRemainingLength + RemainingLength.RemainingLength) > COM.R_BUF.SIZE THEN
							NeedBufferMove := TRUE;
						END_IF
					END_IF	
					IF RemainingLength.RemainingLength > TRANSMIT_BUFFER_SIZE THEN
						//packet needs to be moved into big receive buffer
						SplitPublishLength := RemainingLength.RemainingLength + RemainingLength.SizeRemainingLength + 1;//one byte for fixed packed header
						SplitPublishBufferSize := COM.R_BUF.SIZE - IdxIn;//new splited publish
						MEM.MemMove(pSource:= ADR(COM.R_BUF.BUFFER[IdxIn]), pDestination:= SplitPublishBuffer, uiNumberOfBytes:= UDINT_TO_UINT(SplitPublishBufferSize));
						//clear in Buffer
						COM.R_BUF.SIZE := 0;
						COM.MQTT_RCV_STATE := BYTE#0;//receive zurücksetzten	
						PublishSplited := TRUE;
						CheckLenghtBuffer := TRUE; 	
						PushError(newError:= ERRORS.MOVED_TO_BIG_RECEIVE_BUFFER , text:='');
					END_IF
				END_IF
			END_IF
		END_IF
	MESSAGETYPE.PUBREL:
		IF IdxIn + SIZE_PUBREL > COM.R_BUF.SIZE THEN
			NeedBufferMove := TRUE;
		END_IF
	MESSAGETYPE.UNSUBACK:
		IF IdxIn + SIZE_UNSUBACK > COM.R_BUF.SIZE THEN
			NeedBufferMove := TRUE;
		END_IF
	MESSAGETYPE.SUBACK:
		IF IdxIn + SIZE_SUBACK > COM.R_BUF.SIZE THEN
			NeedBufferMove := TRUE;
		END_IF
	MESSAGETYPE.PUBACK:
		IF IdxIn + SIZE_PUBACK > COM.R_BUF.SIZE THEN
			NeedBufferMove := TRUE;
		END_IF
	MESSAGETYPE.PUBREC:
		IF IdxIn + SIZE_PUBREC > COM.R_BUF.SIZE THEN
			NeedBufferMove := TRUE;
		END_IF
	MESSAGETYPE.PUBCOMP:
		IF IdxIn + SIZE_PUBCOMP > COM.R_BUF.SIZE THEN
			NeedBufferMove := TRUE;
		END_IF

END_CASE

IF NeedBufferMove AND NOT ( IdxIn = 0)THEN
	IF LogBufferMoves THEN
		PushError(newError:= ERRORS.NEED_BUFFER_MOV, text:='');
	END_IF
	MoveBufferForSplitPaket(idx:= IdxIn);
	InBufferMoved := 1;
	
ELSE
	InBufferMoved := 0;
	CountWaitForRestOfPaket := 0;
END_IF

CheckLenghtBuffer := NeedBufferMove;

IF InBufferMoved = 1 THEN
	CountWaitForRestOfPaket := CountWaitForRestOfPaket + 1;
END_IF

IF CountWaitForRestOfPaket > 1000 THEN
	//waited long for rest of paket, so reset...	
	//unknown paket, reset buffer....
	//standard wants to disconnect....
	{info 'TODO:check to make disconnect as parameter'}
	DoDisconnect := TRUE;
	PushError(newError:= ERRORS.FULL_PACKET_NOT_RECEIVED, text:='');
	COM.R_BUF.SIZE := 0;	
	//unknown paket received
	NotKnownPaket := COM.R_BUF.BUFFER[0] AND 16#F0;
	//allway reset receive!
	COM.MQTT_RCV_STATE := BYTE#0;//receive zurücksetzten
	COM.R_BUF.SIZE := 0;
	CountWaitForRestOfPaket := 0;
	CountResetBufferIn := CountResetBufferIn + 1;
END_IF
END_METHOD

METHOD FB_Exit : BOOL 
VAR_INPUT 
 bInCopyCode : BOOL; // TRUE: the exit method is called in order to leave the instance which will be copied afterwards (online change). 
END_VAR
destroy();
END_METHOD

METHOD destroy : bool
VAR_INPUT
END_VAR
VAR
	iu:UINT;
END_VAR
MySplitTopic.destroy();
GVL_MQTT.ProgNum := PROG_NUM.DESTROY_HANDLE_MQTT;
{info 'semaphore'}
IF NOT StepInitDone THEN RETURN;END_IF
//THIS^.DynMemUsagePointer^ := THIS^.DynMemUsagePointer^ - SplitPublishBufferAllocationSize;
DynMemUsagePointer^ := DynMemUsagePointer^ - SplitPublishBufferAllocationSize;
{warning disable C0033}
__DELETE(SplitPublishBuffer);
{warning restore C0033}
StepInitDone := FALSE;
GVL_MQTT.ProgNum := PROG_NUM.DESTROY_HANDLE_MQTT_DONE;
END_METHOD

METHOD OutputPublish
VAR_INPUT
	
	PayloadSize:UDINT;
	//be aware, don't use network buffer, IP_CONTROL may change content
	PayloadPos:POINTER TO BYTE;
	TopicSize:UDINT;
	//be aware, don't use network buffer, IP_CONTROL may change content, must be zero terminated!
	TopicPos:POINTER TO BYTE;
	MQTT_IN_OUT : POINTER TO MQTT_IN_OUT;
	//data must be moved from network buffer to local buffer, doesn't needs to be done, output by callback
	//NeedMove: BOOL;
END_VAR
VAR
	i:UINT;
	match:TOPIC_MATCH;
	PointerToSplit: POINTER TO SPLIT_TOPIC;
	DataForCallback:CALLBACK_DATA;
END_VAR
//here make everything to give out publish, and test if topic fits to my borders...
CountOutputPublishCalled := CountOutputPublishCalled + 1;
IF MySplitTopic.NewTopic(in:= TopicPos, test := FALSE, SizeOfString:= UDINT_TO_UINT(TopicSize)) = TOPIC_VALID.TOPIC_NOT_VALID THEN
	//topic is not in my borders so throw away data...
	{info 'configure to disconnect?'}
	{ info 'make count var...'}
	CountSplitTopicSizeExceeded := CountSplitTopicSizeExceeded + 1;
	RETURN;
END_IF
//now search the right callback and call it...
PointerToSplit := MySplitTopic.GetSplitTopic();
DataForCallback.Payload := PayloadPos;
DataForCallback.PayloadSize := PayloadSize;
DataForCallback.PayloadString :=PayloadPos;
DataForCallback.TopicOut := TopicPos;
DataForCallback.TopicOutSplit := PointerToSplit;
DataForCallback.PayloadIsString := SubscribeCallbacks[i].ExpectingString;

FOR i := 0 TO CALLBACKS_BUFFER_SIZE - 1 DO
	IF NOT SubscribeCallbacks[i].free THEN
		match := SubscribeCallbacks[i].SplitTopic^.CheckTopicMatchToMe(with:=PointerToSplit);
		IF match = TOPIC_MATCH.TOPIC_MATCHES THEN
			SubscribeCallbacks[i].Callback.PublishReceived(Data:=DataForCallback);
		END_IF
	END_IF
END_FOR
END_METHOD

METHOD MergeSplitedPublish
VAR_INPUT
	MQTT_IN_OUT: POINTER TO MQTT_IN_OUT;
END_VAR
VAR
	BytesToMove : UINT;
END_VAR
//move every new data to publish receive buffer untill all data is received
BytesToMove := TO_UINT(MIN(com.R_BUF.SIZE, SplitPublishLength - SplitPublishBufferSize));
MEM.MemMove(pSource:= ADR(COM.R_BUF.BUFFER), pDestination:= ADR(SplitPublishBuffer[SplitPublishBufferSize]), uiNumberOfBytes:= BytesToMove);
SplitPublishBufferSize := SplitPublishBufferSize + BytesToMove;
IF SplitPublishBufferSize >= SplitPublishLength THEN
	//SplitPublishLock := TRUE;
	PublishSplited := FALSE;
	//ParsePublish will insert string termination if no network buffer
	ParseIncomingPublish(
	MQTT_IN_OUT:= MQTT_IN_OUT, 
	idx:= 0, 
	BufferIn:= SplitPublishBuffer, 
	BufferSize:= SplitPublishBufferSize,
	NetworkBuffer := FALSE);
END_IF
//check if there is more data in buffer --> new packet
IF BytesToMove < COM.R_BUF.SIZE THEN
	//move buffer and set new size...
	MEM.MemMove(pSource:= ADR(COM.R_BUF.BUFFER[BytesToMove]), pDestination:= ADR(COM.R_BUF.BUFFER),
				uiNumberOfBytes:= COM.R_BUF.SIZE - BytesToMove);
	COM.R_BUF.SIZE := COM.R_BUF.SIZE - BytesToMove;
ELSE
	//clear buffer
	COM.R_BUF.SIZE := 0;
	COM.MQTT_RCV_STATE := BYTE#0;//receive zurücksetzten	
END_IF
END_METHOD

METHOD Publish : BOOL
VAR_INPUT
	data : POINTER TO DATA_TO_BROKER;
END_VAR
VAR
	i:UINT;
END_VAR
Publish := FALSE;
if not connected then return; end_if
FOR i := 0 TO MyConstants.IN_OUT_SLOTS_SIZE - 1 DO
	IF OutDataSlots[i].step = STEPS_OUT.WAIT_DATA THEN
		OutDataSlots[i].InDataFromFb := data;//set Data
		//Pakte id = slot + 1....
		OutDataSlots[i].InDataFromFb^.PaketId := i + 1;
		OutgoingPublishOrderIndexCounter := OutgoingPublishOrderIndexCounter + 1;
		OutDataSlots[i].PUBLISHOrder :=  OutgoingPublishOrderIndexCounter;
		OutDataSlots[i].step := STEPS_OUT.SEND_PUBLSIH;
		CountSendedPublishs := CountSendedPublishs + 1;
		CounterPublishSendForMonitor := CounterPublishSendForMonitor + 1;
		OutDataSlots[i].PUBRELRepeatCounter := 0;
		Publish := TRUE;
		EXIT;
	END_IF
END_FOR

IF NOT Publish THEN
	PushError(newError:= ERRORS.PUBLISH_NO_SLOT_FREE, text:='');
END_IF
END_METHOD

METHOD PublishSendDone
VAR_INPUT
	slot:POINTER TO MQTT_OUT_DATA;
END_VAR
slot^.TimeOutStarted := TRUE;//start Timeout
CASE slot^.InDataFromFb^.MessageQoS OF
	QoS.AtMostOnce:
	//paket gone and bye bye, on QoS 0 
	slot^.InDataFromFb^.SendSucsess := TRUE;
	slot^.step := STEPS_OUT.WAIT_DATA;//can get new data
	QoS.AtLeastOnce:
		slot^.step := STEPS_OUT.WAIT_PUBACK;//wait for ACK
		IF NOT slot^.InDataFromFb^.DUP THEN
			Publishsunacknowledged := Publishsunacknowledged + 1;
		END_IF
	QoS.ExactlyOnce:
		slot^.step := STEPS_OUT.WAIT_PUBREC;//wait for REC
		IF NOT slot^.InDataFromFb^.DUP THEN
			Publishsunacknowledged := Publishsunacknowledged + 1;
		END_IF
END_CASE
END_METHOD

METHOD PushError
VAR_INPUT
	newError:ERRORS;
	text:STRING(255);
END_VAR
VAR
	i:UINT;
	cleanError:ONE_ERROR ;
END_VAR
//move all Errors...

FOR i:= COUNT_ERROR_HISTORY - 1 TO 1 BY - 1  DO
	ErrorHistory[i] := ErrorHistory[i - 1];
END_FOR
ErrorHistory[0] := cleanError;
ErrorHistory[0].error  := newError;
ErrorHistory[0].when := localTdi.SYSTEM_TIME;
ErrorHistory[0].text := text;
ErrorHistory[0].MqttsDoneIo := MqttsDoneIo;
ErrorHistory[0].ReceivedBytes := ReceivedBytes;
ErrorHistory[0].SendetBytes := SendetBytes;

IF newError = ERRORS.CONNECTION_REFUSED THEN
	ErrorHistory[0].ERROR_C := COM.ERROR_C;
	ErrorHistory[0].ERROR_T := COM.ERROR_T;
END_IF
END_METHOD

END_FUNCTION_BLOCK

// MQTT/Function Blocks/InsertSplitTopic
FUNCTION_BLOCK InsertSplitTopic
VAR_INPUT
	//topic to insert....
	topic:POINTER TO STRING;
	//length of topic
	len:UINT;
	//address to buffer
	buff:POINTER TO BYTE;
	//Start to insert
	pos:UINT;
	//size of buffer
	size:UINT;
	
END_VAR
VAR_OUTPUT
	state : INSERT_SPLIT_RETURN;
	new_pos:UINT;
END_VAR
VAR
	step: INT;
	akt_pos:UINT;
END_VAR
VAR_TEMP
	
	bytes_to_send:UINT;
END_VAR

//always make my output valid
new_pos := pos;

IF step = 0 THEN
	step := 10;//start insert...
END_IF

//don't use case, so save a cyle...
IF step = 10 THEN
	//check if buffer size is enough for header
	IF size - new_pos < 2 THEN
		state := INSERT_SPLIT_RETURN.INSERT_ERROR;
		RETURN;
	END_IF
	buff[new_pos]:= OSCAT_BASIC.BYTE_OF_DWORD(in:= len, N:= 1);
	buff[new_pos+1]:= OSCAT_BASIC.BYTE_OF_DWORD(in:= len, N:= 0);
	new_pos := new_pos + 2;
	step := 20;
END_IF

IF step = 20 THEN
	//evaluate if we have to split topic....
	IF size - pos < len THEN
		step := 30;
		akt_pos := 0;
	ELSE
		//here no split needed
		MEM.MemMove(pSource:= topic, pDestination:= ADR(buff[new_pos]), uiNumberOfBytes:= len);
		new_pos := new_pos + len;//new pos for output
		state := INSERT_SPLIT_RETURN.INSERT_DONE;
		step := 0;
	END_IF
END_IF

IF step = 30 THEN
	//now do split topic...
	bytes_to_send := MIN(size - new_pos, len - akt_pos);
	MEM.MemMove(pSource:= ADR(topic^[akt_pos]), pDestination:= ADR(buff[new_pos]), uiNumberOfBytes:= bytes_to_send);
	akt_pos := akt_pos + bytes_to_send;
	new_pos := new_pos +  bytes_to_send;
	IF akt_pos + 1 >= len THEN
		//send done
		state := INSERT_SPLIT_RETURN.INSERT_DONE;
		step := 0;
	ELSE
		state := INSERT_SPLIT_RETURN.INSERT_PENDING;
	END_IF
END_IF

METHOD reset
VAR_INPUT
END_VAR
step := 0;
END_METHOD

END_FUNCTION_BLOCK

// MQTT/Function Blocks/InsertSplitPayload
FUNCTION_BLOCK InsertSplitPayload
VAR_INPUT
	//payload to insert....
	payload:POINTER TO BYTE;
	//length of payload
	len:UDINT;
	//address to buffer
	buff:POINTER TO BYTE;
	//Start to insert
	pos:UINT;
	//size of buffer
	size:UINT;
	
END_VAR
VAR_OUTPUT
	state : INSERT_SPLIT_RETURN;
	new_pos:UINT;
END_VAR
VAR
	step: INT;
	akt_pos:UDINT;
END_VAR
VAR_TEMP
	
	bytes_to_send:UINT;
END_VAR

//always make my output valid
new_pos := pos;

IF step = 0 THEN
	step := 10;//start insert...
END_IF

//don't use case, so save a cyle...
IF step = 10 THEN
	//evaluate if we have to split payload....
	IF size - pos < len THEN
		step := 20;
		akt_pos := 0;
	ELSE
		//here no split needed
		MEM.MemMove(pSource:= payload, pDestination:= ADR(buff[new_pos]), uiNumberOfBytes:= UDINT_TO_UINT(len));
		new_pos := UDINT_TO_UINT(new_pos + len);//new pos for output
		state := INSERT_SPLIT_RETURN.INSERT_DONE;
		step := 0;
	END_IF
END_IF

IF step = 20 THEN
	//now do split payload...
	bytes_to_send := UDINT_TO_UINT(MIN(size - new_pos, len - akt_pos));
	MEM.MemMove(pSource:= ADR(payload[akt_pos]), pDestination:= ADR(buff[new_pos]), uiNumberOfBytes:= bytes_to_send);
	akt_pos := akt_pos + bytes_to_send;
	new_pos := new_pos +  bytes_to_send;
	IF akt_pos + 1 >= len THEN
		//send done
		state := INSERT_SPLIT_RETURN.INSERT_DONE;
		step := 0;
	ELSE
		state := INSERT_SPLIT_RETURN.INSERT_PENDING;
	END_IF
END_IF

METHOD reset
VAR_INPUT
END_VAR
step := 0;
END_METHOD

END_FUNCTION_BLOCK

// MQTT/Function Blocks/MQTT_CONTROL

(*
Controls send and receive to an MQTT broker
*)

FUNCTION_BLOCK MQTT_CONTROL

VAR_IN_OUT
	COM : MQTT_COM;
	INFO : MQTT_INFO;
END_VAR
VAR_OUTPUT
END_VAR
VAR
	IP_C : IP_C;
	URL_DATA : url;
	
	IPC :CommonTypesAndFunctions.IP_CONTROL_TLS;
	sResultIP : STRING; // IP-Address behind hostname
	rtsResult : RTS_IEC_RESULT;
	step : INT;
	snd_step : INT;
	TON_WAIT : OSCAT_BASIC.TON;
	last_step : INT;
	idx1 : UINT;
	connectToLocalhost: BOOL;
	staticIP: BOOL;

	timeout1 : TIME;
	timeout2 : TIME;
	ip_c_red_disable : BOOL;
	remaining_length:UINT;
	domainLowercase:STRING(255);

	(*
	LOG_MSG : LOG_MSG;
	_debug_enable : BOOL := TRUE;
	*)
	nop: INT;
	(********************************************************************************)
	//here all TLS Stuff
	
	S_BUF : NETWORK_BUFFER;
	R_BUF : NETWORK_BUFFER;
	
	(********************************************************************************)
	
	
	TLSConnection: RTS_IEC_HANDLE;
END_VAR

IF com.ERROR_C <> 0 THEN
 step := step;
END_IF 
//init Pointers


CASE step OF

00:	IF COM.MQTT_CON THEN

		timeout1 := MAX(T#10S,COM.TIMEOUT);
		timeout2 := timeout1 + T#1s;
		INFO.MQTT_ERROR := '';
		COM.ERROR_C := DWORD#0;
		COM.ERROR_T := BYTE#0;
		URL_DATA := STRING_TO_URL(STR:=COM.MQTT_URL,DEFAULT_PROTOCOL:='',DEFAULT_PATH:='/');
		domainLowercase := OSCAT_BASIC.LOWERCASE(str:=URL_DATA.DOMAIN );
		IF  CommonTypesAndFunctions.StrEqualsAtStart(str1:= ADR(domainLowercase), str2:= ADR('localhost')) THEN
			connectToLocalhost := TRUE;
		ELSE
			connectToLocalhost := FALSE;
		END_IF
		IF OSCAT_NETWORK.IP4_DECODE(str:= URL_DATA.DOMAIN) > 0 THEN
			sResultIP := URL_DATA.DOMAIN;
			staticIP := TRUE;
		ELSE
			staticIP := FALSE;
		END_IF
		IF connectToLocalhost OR staticIP THEN
			//jump to connect
			step := 20;
		ELSE
			//get ip by dns
			step := 10;
		END_IF
	END_IF;

10:
	IF CommonTypesAndFunctions.ResolveIPAddr(sHost:= URL_DATA.DOMAIN, sIPResult:= ADR(sResultIP)) = CmpErrors.Errors.ERR_OK THEN
		step := 20;
	ELSE
		step := 980;
	END_IF

20:	(* MQTT Steuerkanal einrichten *)
	IF URL_DATA.PORT = WORD#0 THEN
		URL_DATA.PORT := WORD#1883; (* Standard Port *)
	END_IF;
	IP_C.C_PORT := URL_DATA.PORT; (* Portnummer eintragen *)
	IF connectToLocalhost THEN
		IP_C.C_IP := IP4_DECODE('127.0.0.1'); (* IP eintragen, localhost *)
	ELSE
		IP_C.C_IP := IP4_DECODE(sResultIP); (* IP eintragen *)
	END_IF
  	
	IP_C.C_MODE := BYTE#0; (* Mode: TCP+ACTIV+PORT *)
  	IP_C.TIME_RESET := TRUE; (* Zeitueberwachung rücksetzen *)
  	IP_C.C_ENABLE := TRUE; (* Verbindungsaufbau freigeben *)
  	IP_C.R_OBSERVE := FALSE; (* Empfangsueberwachung *)
	COM.R_BUF.SIZE := UINT#0;
	COM.MQTT_RCV_STATE := BYTE#0;
	step := 30;
	

30:	 IF IP_C.C_STATE = BYTE#255 THEN
		COM.S_BUF.BUFFER[0] := MESSAGETYPE.CONNECT;
		COM.S_BUF.BUFFER[1] := 0;//Header length, cal at least
		COM.S_BUF.BUFFER[2] := 0;//Variable Header length
		COM.S_BUF.BUFFER[3] := 4;//Variable Header length
		COM.S_BUF.BUFFER[4] := OSCAT_BASIC.CODE(STR:= 'M', POS:= 1);//Protokoll name
		COM.S_BUF.BUFFER[5] := OSCAT_BASIC.CODE(STR:= 'Q', POS:= 1);//Protokoll name
		COM.S_BUF.BUFFER[6] := OSCAT_BASIC.CODE(STR:= 'T', POS:= 1);//Protokoll name
		COM.S_BUF.BUFFER[7] := OSCAT_BASIC.CODE(STR:= 'T', POS:= 1);//Protokoll name
		COM.S_BUF.BUFFER[8] := 4; //Protokoll Level
		COM.S_BUF.BUFFER[9] := 2#00110110;//Connect flags
							   //|||||||+-Reserved
							   //||||||+--Clean Session
							   //|||||+---Will Flag
							   //|||++----Will QoS
							   //||+------Will Retain
							   //|+-------Password Flag
							   //+--------UserNameFlag
		COM.S_BUF.BUFFER[10] := OSCAT_BASIC.BYTE_OF_DWORD(in:= MyConstants.KEEP_ALIVE_TIME, N:= 1);//keep alive MSB
		COM.S_BUF.BUFFER[11] := OSCAT_BASIC.BYTE_OF_DWORD(in:= MyConstants.KEEP_ALIVE_TIME, N:= 0);//keep alive LSB
		//idx1 points to next free byte
		//now put in client id 
		idx1 := InsertStringToBufferAndLength(Str:= ADR(COM.CLIENT_ID), buff:= ADR(COM.S_BUF.BUFFER), pos:= 12(*, size:= OSCAT_NETWORK.Constants.NETWORK_BUFFER_LONG_SIZE*));
		//now put in will topic
		//WillTopic := Standard.CONCAT(STR1:= COM.CLIENT_ID, STR2:= Standard.CONCAT(STR1:= '/', STR2:= COM.CLIENT_WILL_TOPIC));
		idx1 := InsertStringToBufferAndLength(Str:= ADR(COM.CLIENT_WILL_TOPIC), buff:= ADR(COM.S_BUF.BUFFER), pos:= idx1(*, size:= OSCAT_NETWORK.Constants.NETWORK_BUFFER_LONG_SIZE*));
		//now put in will message
		//IF Standard.LEN(STR:= COM.CLIENT_WILL_MESSAGE_DEAD) > 0 THEN
		idx1 := InsertStringToBufferAndLength(Str:= ADR(COM.CLIENT_WILL_MESSAGE_DEAD), buff:= ADR(COM.S_BUF.BUFFER), pos:= idx1(*, size:= OSCAT_NETWORK.Constants.NETWORK_BUFFER_LONG_SIZE*));
		//END_IF
		//if user is given, set user bit an insert username
		IF Standard.LEN(STR:= URL_DATA.USER) > 0 THEN
			COM.S_BUF.BUFFER[9] := COM.S_BUF.BUFFER[9] OR 2#10000000;
			//now put in user name
			idx1 := InsertStringToBufferAndLength(Str:= ADR(URL_DATA.USER), buff:= ADR(COM.S_BUF.BUFFER), pos:= idx1(*, size:= OSCAT_NETWORK.Constants.NETWORK_BUFFER_LONG_SIZE*));
		END_IF
		//if password is given, set password bit an insert username
		IF Standard.LEN(STR:= URL_DATA.PASSWORD) > 0 THEN
			COM.S_BUF.BUFFER[9] := COM.S_BUF.BUFFER[9] OR 2#1000000;
			//now put in user name
			idx1 := InsertStringToBufferAndLength(Str:= ADR(URL_DATA.PASSWORD), buff:= ADR(COM.S_BUF.BUFFER), pos:= idx1(*, size:= OSCAT_NETWORK.Constants.NETWORK_BUFFER_LONG_SIZE*));
		END_IF
		//now cal packet lengt and insert remaining legth
		remaining_length := idx1 - 2;
		DoRemainingLength(buffer:= ADR(com.S_BUF.BUFFER), RemainingLength:= remaining_length);
		//now send data
		COM.S_BUF.SIZE := idx1;
		step := 40;//wait for CONNACK
	END_IF
	
		
40:	//IF COM.MQTT_RCV_STATE = BYTE#1 THEN//received packet
	IF COM.R_BUF.SIZE > 0 THEN//received packet
		IF COM.R_BUF.BUFFER[0] <> MESSAGETYPE.CONNACK THEN
			step := 700;//close connection
		ELSE//get connack packet
			IF COM.R_BUF.BUFFER[3] = 0 THEN
				//connection accepted
				INFO.MQTT_CONNECTED := TRUE;
				COM.R_BUF.SIZE := 0;
				COM.MQTT_RCV_STATE := BYTE#0;
				step := 300;
			ELSE
				step := 700;//close connection
			END_IF
		END_IF
		
	END_IF


(* ================================================== *)

300:	step := UINT_TO_INT(SEL(COM.MQTT_CON,700,310)); (* Schritt-Selektion *)

310:	step := 300; (* dummy step *)

(* ================================================== *)

700: (* COM_QUIT *)
	//INFO.MQTT_CONNECTED := FALSE;
	IF COM.MQTT_ABORT THEN
		step := 980;//close without disconnect packet
		COM.MQTT_ABORT := FALSE;
	ELSE
		COM.S_BUF.BUFFER[0] := MESSAGETYPE.DISCONNECT; (* 0x01 COM_QUIT mqtt_close *)
		COM.S_BUF.BUFFER[1] := 0;
		COM.S_BUF.SIZE := UINT#2; (* Sendelänge eintragen *)
		
		ip_c_red_disable := TRUE;
		step := 710;
	END_IF
710:	IF COM.S_BUF.SIZE = BYTE#0 THEN (* letztes Paket gesendet?*)
		step := 980;
	END_IF;

(* ================================================== *)

980:IP_C.C_ENABLE := FALSE; (* MQTT Steuerkanal schliessen *)
	ip_c_red_disable := FALSE;
	INFO.MQTT_CONNECTED := FALSE;
	COM.MQTT_CON := FALSE;
	COM.S_BUF.SIZE := UINT#0;
	COM.R_BUF.SIZE := UINT#0;
	snd_step := 0;
	step := 990;
	(*####################  DEBUG-MESSAGE  ###################################*)
	(*IF _debug_enable THEN
		LOG_CL.NEW_MSG := 'QUIT: ERROR CODE >~1< TYPE >~2<';
		LOG_CL.PRINTF[1] := DWORD_TO_STRH(COM.ERROR_C);
		LOG_CL.PRINTF[2] := BYTE_TO_STRING(COM.ERROR_T);
		LOG_MSG();
	END_IF;*)
	(*########################################################################*)

990:IF IP_C.C_STATE = BYTE#0 THEN
		step := 0;
	END_IF;

END_CASE;

(* ++++++++++++++++++++++++++++++++++++++++++++++++++++++++++ *)
IF step > 40 THEN
	IF COM.R_BUF.SIZE >= UINT#1 THEN (* Daten wurden empfangen ? neue kommunikation*)
		
		COM.MQTT_RCV_STATE := BYTE#1;
		
	END_IF;
END_IF;
(* automatisches Datensenden *)

CASE snd_step OF

00:	IF step > 40 THEN
	
		IF COM.S_BUF.SIZE > UINT#0 THEN
	
		    (*####################  DEBUG-MESSAGE  ###################################*)
	        (*IF _debug_enable THEN
	          LOG_CL.NEW_MSG := 'SND: size >~1<';
	          LOG_CL.PRINTF[1] := UINT_TO_STRING(COM.S_BUF.SIZE);
	          LOG_MSG();
	        END_IF;*)
	        (*########################################################################*)

			snd_step := 10;
		END_IF;		
	END_IF;

10:	IF COM.S_BUF.SIZE = UINT#0 THEN (* warten bis alle daten gesendet sind *)
		snd_step := 0;
	END_IF;

END_CASE;

(* Globale Fehlerbehandlung für Haupt-Routine *)
IF COM.ERROR_T = BYTE#0 AND step > 20 THEN (* noch kein Fehler gespeichert und Hauptroutine aktiv *)
	IF IP_C.ERROR > DWORD#0 AND IP_C.C_ENABLE AND NOT IP_C.TIME_RESET THEN  (* IP Control *)
		IF ip_c_red_disable = FALSE OR IP_C.ERROR <> DWORD#16#FD000000 THEN
			COM.ERROR_C := IP_C.ERROR;
			COM.ERROR_T := BYTE#2;
			step := 980;
		END_IF;
	END_IF;
END_IF;

IF TON_WAIT.Q THEN (* Ablaufstörung - Schrittkette *)
	COM.ERROR_C := INT_TO_DWORD(step); (* aktuellen Schritt eintragen *)
	COM.ERROR_T := BYTE#5;
	step := 980;
END_IF;

(* ######################################################## *)

